KUKA KRL program: MyProgram_049().src

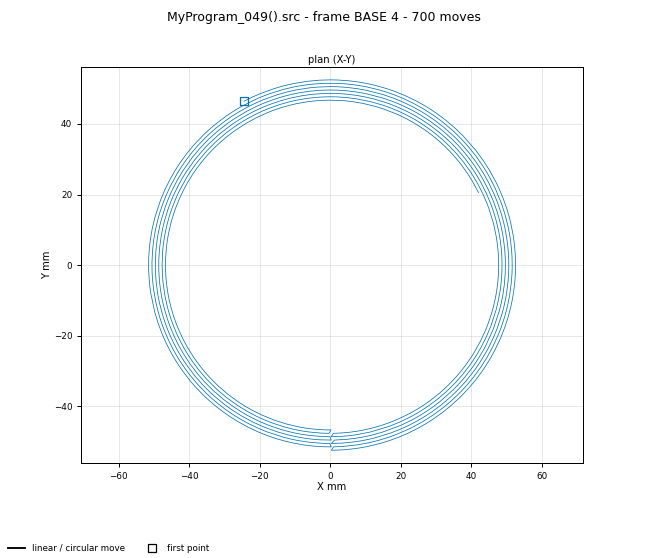
[picture p0: tool path of MyProgram_049().src in frame BASE 4, 700 of 700 moves have a stored position in this frame; points joined in program order, loops and branches not executed]
&ACCESS RVP
&REL 1
&PARAM TEMPLATE = C:\KRC\Roboter\Template\vorgabe
&PARAM EDITMASK = *
DEF MyProgram_049()
; ---- Setting reference (Base) ----
$BASE = BASE_DATA[4]

; --------------------------
; ---- Setting tool (TCP) ----
$TOOL = TOOL_DATA[3]
; --------------------------

$VEL.CP = VEL_APROX_PRINT
Startdeposition()
$VEL.CP = VEL_PRINT
LIN {X -24.4251,Y 46.489,Z 66,A 110.3298,B 24.8528,C -2.799,E1 24.9276,E2 -26.6779} C_DIS
LIN {X -22.2975,Y 47.5462,Z 66,A 107.8402,B 24.8522,C -2.8046,E1 24.9338,E2 -24.1953} C_DIS
LIN {X -20.0444,Y 48.539,Z 66,A 104.5324,B 24.8529,C -2.7984,E1 24.9424,E2 -20.8649} C_DIS
LIN {X -15.8817,Y 50.0558,Z 66,A 100.3319,B 24.8512,C -2.8146,E1 24.9534,E2 -16.695} C_DIS
LIN {X -13.4432,Y 50.7654,Z 66,A 97.3988,B 24.8512,C -2.8147,E1 24.9613,E2 -13.7577} C_DIS
LIN {X -10.7407,Y 51.4051,Z 66,A 93.9354,B 24.8517,C -2.8101,E1 24.9708,E2 -10.279} C_DIS
LIN {X -6.5682,Y 52.1029,Z 66,A 89.9124,B 24.8503,C -2.8232,E1 24.9818,E2 -6.2837} C_DIS
LIN {X -3.1559,Y 52.4207,Z 66,A 85.9853,B 24.8504,C -2.8216,E1 24.9927,E2 -2.3511} C_DIS
LIN {X 0.019,Y 52.5158,Z 66,A 82.4303,B 24.8505,C -2.8209,E1 25.0027,E2 1.2058} C_DIS
LIN {X 2.2082,Y 52.4685,Z 66,A 79.9006,B 24.8507,C -2.8187,E1 25.0097,E2 3.7403} C_DIS
LIN {X 5.4247,Y 52.234,Z 66,A 76.6583,B 24.8503,C -2.8233,E1 25.0187,E2 6.9698} C_DIS
LIN {X 8.0055,Y 51.9012,Z 66,A 73.774,B 24.8504,C -2.8218,E1 25.0267,E2 9.8551} C_DIS
LIN {X 10.5647,Y 51.4413,Z 66,A 71.0397,B 24.8504,C -2.8225,E1 25.0342,E2 12.5846} C_DIS
LIN {X 12.7838,Y 50.935,Z 66,A 68.4031,B 24.8508,C -2.8183,E1 25.0414,E2 15.2272} C_DIS
LIN {X 15.987,Y 50.0225,Z 66,A 65.1391,B 24.8503,C -2.8226,E1 25.0501,E2 18.4755} C_DIS
LIN {X 18.0888,Y 49.3014,Z 66,A 62.3939,B 24.8512,C -2.8145,E1 25.0573,E2 21.2343} C_DIS
LIN {X 21.2443,Y 48.026,Z 66,A 58.6048,B 24.8518,C -2.8092,E1 25.0671,E2 25.0269} C_DIS
LIN {X 24.339,Y 46.5341,Z 66,A 55.5963,B 24.8507,C -2.8188,E1 25.0745,E2 28.0049} C_DIS
LIN {X 26.498,Y 45.3396,Z 66,A 52.1536,B 24.8527,C -2.8006,E1 25.083,E2 31.4803} C_DIS
LIN {X 28.6427,Y 44.0153,Z 66,A 49.6719,B 24.8526,C -2.8016,E1 25.0888,E2 33.9516} C_DIS
LIN {X 30.216,Y 42.9521,Z 66,A 47.4699,B 24.8532,C -2.7957,E1 25.0939,E2 36.1601} C_DIS
LIN {X 32.4632,Y 41.2792,Z 66,A 44.4209,B 24.8537,C -2.7905,E1 25.1006,E2 39.2102} C_DIS
LIN {X 35.455,Y 38.7397,Z 66,A 40.2431,B 24.8544,C -2.7844,E1 25.1094,E2 43.3862} C_DIS
LIN {X 37.586,Y 36.6762,Z 66,A 36.7099,B 24.8557,C -2.7718,E1 25.1164,E2 46.9343} C_DIS
LIN {X 41.2065,Y 32.5552,Z 66,A 31.7321,B 24.855,C -2.7786,E1 25.1255,E2 51.8734} C_DIS
LIN {X 43.4466,Y 29.4994,Z 66,A 26.8425,B 24.8576,C -2.7532,E1 25.1335,E2 56.7995} C_DIS
LIN {X 45.1779,Y 26.7727,Z 66,A 23.6494,B 24.8579,C -2.7509,E1 25.1382,E2 59.9819} C_DIS
LIN {X 47.1008,Y 23.2237,Z 66,A 19.3403,B 24.8589,C -2.741,E1 25.1439,E2 64.2916} C_DIS
LIN {X 47.7499,Y 21.8578,Z 66,A 16.8923,B 24.8611,C -2.72,E1 25.1467,E2 66.7761} C_DIS
LIN {X 48.9324,Y 19.0647,Z 66,A 14.0783,B 24.861,C -2.7208,E1 25.1497,E2 69.5726} C_DIS
LIN {X 50.0654,Y 15.8514,Z 66,A 10.5617,B 24.8616,C -2.7142,E1 25.1528,E2 73.0851} C_DIS
LIN {X 50.6849,Y 13.7421,Z 66,A 8.1164,B 24.8625,C -2.7061,E1 25.1547,E2 75.5356} C_DIS
LIN {X 51.1251,Y 12.0025,Z 66,A 5.8316,B 24.8638,C -2.6933,E1 25.1562,E2 77.8373} C_DIS
LIN {X 51.8393,Y 8.4,Z 66,A 2.4748,B 24.8636,C -2.6947,E1 25.1579,E2 81.1712} C_DIS
LIN {X 52.1505,Y 6.1764,Z 66,A -0.4769,B 24.8655,C -2.6766,E1 25.1589,E2 84.1483} C_DIS
LIN {X 52.4193,Y 3.1759,Z 66,A -3.9297,B 24.8669,C -2.6628,E1 25.1596,E2 87.6132} C_DIS
LIN {X 52.5126,Y -0.462,Z 66,A -7.4944,B 24.8672,C -2.6589,E1 25.1597,E2 91.1659} C_DIS
LIN {X 52.4191,Y -3.1656,Z 66,A -10.1321,B 24.8675,C -2.6562,E1 25.1594,E2 93.7943} C_DIS
LIN {X 52.2992,Y -4.7558,Z 66,A -12.1864,B 24.8687,C -2.6441,E1 25.1589,E2 95.8651} C_DIS
LIN {X 51.9991,Y -7.3421,Z 66,A -14.8639,B 24.8693,C -2.6386,E1 25.158,E2 98.5398} C_DIS
LIN {X 51.6388,Y -9.5543,Z 66,A -17.2732,B 24.87,C -2.6316,E1 25.1568,E2 100.9514} C_DIS
LIN {X 51.2544,Y -11.4372,Z 66,A -19.8065,B 24.8715,C -2.6159,E1 25.1553,E2 103.5072} C_DIS
LIN {X 50.3186,Y -15.0287,Z 66,A -23.5172,B 24.8721,C -2.6105,E1 25.1526,E2 107.2093} C_DIS
LIN {X 49.5084,Y -17.5135,Z 66,A -26.3955,B 24.873,C -2.6012,E1 25.15,E2 110.0933} C_DIS
LIN {X 48.4841,Y -20.1769,Z 66,A -29.1133,B 24.873,C -2.6002,E1 25.1472,E2 112.7985} C_DIS
LIN {X 47.9293,Y -21.4606,Z 66,A -31.0442,B 24.8743,C -2.5872,E1 25.145,E2 114.7498} C_DIS
LIN {X 46.529,Y -24.3487,Z 66,A -34.3749,B 24.875,C -2.5805,E1 25.1408,E2 118.0783} C_DIS
LIN {X 45.286,Y -26.5899,Z 66,A -37.4931,B 24.8764,C -2.5659,E1 25.1365,E2 121.2151} C_DIS
LIN {X 43.7354,Y -29.0701,Z 66,A -40.2741,B 24.8764,C -2.5655,E1 25.1323,E2 123.9829} C_DIS
LIN {X 42.5013,Y -30.8459,Z 66,A -42.7432,B 24.8773,C -2.5569,E1 25.1283,E2 126.4603} C_DIS
LIN {X 41.2562,Y -32.4924,Z 66,A -45.0593,B 24.878,C -2.5497,E1 25.1243,E2 128.7827} C_DIS
LIN {X 39.4232,Y -34.6939,Z 66,A -48.1201,B 24.8786,C -2.5431,E1 25.1188,E2 131.8452} C_DIS
LIN {X 36.7356,Y -37.5281,Z 66,A -52.9038,B 24.8806,C -2.5222,E1 25.1093,E2 136.6578} C_DIS
LIN {X 33.9294,Y -40.083,Z 66,A -56.4666,B 24.8804,C -2.5246,E1 25.1019,E2 140.2009} C_DIS
LIN {X 31.7525,Y -41.829,Z 66,A -59.5227,B 24.881,C -2.5179,E1 25.0952,E2 143.2616} C_DIS
LIN {X 29.2965,Y -43.5834,Z 66,A -62.5914,B 24.8812,C -2.5158,E1 25.0882,E2 146.3246} C_DIS
LIN {X 27.1565,Y -44.9481,Z 66,A -65.8284,B 24.8825,C -2.5014,E1 25.0804,E2 149.5854} C_DIS
LIN {X 24.6543,Y -46.3684,Z 66,A -68.7154,B 24.8825,C -2.501,E1 25.0734,E2 152.4651} C_DIS
LIN {X 22.1208,Y -47.6287,Z 66,A -71.7781,B 24.883,C -2.4967,E1 25.0657,E2 155.5301} C_DIS
LIN {X 19.4367,Y -48.7857,Z 66,A -74.9858,B 24.8835,C -2.4918,E1 25.0574,E2 158.7419} C_DIS
LIN {X 16.7705,Y -49.7651,Z 66,A -78.018,B 24.8837,C -2.4891,E1 25.0494,E2 161.7742} C_DIS
LIN {X 14.1882,Y -50.5619,Z 66,A -81.1897,B 24.8844,C -2.4816,E1 25.0409,E2 164.9583} C_DIS
LIN {X 10.6217,Y -51.4296,Z 66,A -84.7511,B 24.884,C -2.4863,E1 25.0312,E2 168.5038} C_DIS
LIN {X 8.5887,Y -51.8079,Z 66,A -87.0096,B 24.8841,C -2.4845,E1 25.025,E2 170.764} C_DIS
LIN {X 6.6367,Y -52.0936,Z 66,A -89.3786,B 24.8846,C -2.4791,E1 25.0184,E2 173.144} C_DIS
LIN {X 3.7845,Y -52.379,Z 66,A -92.2753,B 24.8844,C -2.4818,E1 25.0104,E2 176.0327} C_DIS
LIN {X 1.9687,Y -52.4779,Z 66,A -94.4349,B 24.8848,C -2.4778,E1 25.0043,E2 178.201} C_DIS
LIN {X 0.2751,Y -52.5115,Z 66,A -95.8459,B 24.8841,C -2.4854,E1 25.0004,E2 179.5939} C_DIS
Enddeposition()
LIN {X 0.2751,Y -52.5115,Z 66,A -95.8459,B 24.8841,C -2.4854,E1 25.0004,E2 179.5939} C_DIS
Startdeposition()
$VEL.CP = VEL_PRINT
LIN {X 0.9003,Y -51.5477,Z 66,A -94.1918,B 24.8808,C -2.5197,E1 25.0053,E2 177.8585} C_DIS
LIN {X 3.5763,Y -51.4318,Z 66,A -90.9185,B 24.8802,C -2.5264,E1 25.0144,E2 174.5705} C_DIS
LIN {X 7.7801,Y -50.9656,Z 66,A -86.3222,B 24.8801,C -2.5274,E1 25.0272,E2 169.9756} C_DIS
LIN {X 10.8144,Y -50.4088,Z 66,A -83.1139,B 24.8802,C -2.5261,E1 25.0359,E2 166.7742} C_DIS
LIN {X 13.4755,Y -49.7634,Z 66,A -79.8609,B 24.8795,C -2.5332,E1 25.0448,E2 163.5094} C_DIS
LIN {X 16.9849,Y -48.6775,Z 66,A -76.2382,B 24.8799,C -2.5292,E1 25.0543,E2 159.903} C_DIS
LIN {X 18.7561,Y -48.0231,Z 66,A -73.5337,B 24.8785,C -2.5438,E1 25.0615,E2 157.1698} C_DIS
LIN {X 22.8223,Y -46.2294,Z 66,A -69.2117,B 24.879,C -2.5391,E1 25.0724,E2 152.8697} C_DIS
LIN {X 26.1375,Y -44.4389,Z 66,A -64.44,B 24.8772,C -2.558,E1 25.0841,E2 148.0673} C_DIS
LIN {X 29.0142,Y -42.6165,Z 66,A -60.8596,B 24.8769,C -2.5612,E1 25.0924,E2 144.4913} C_DIS
LIN {X 31.4014,Y -40.8897,Z 66,A -57.7626,B 24.8765,C -2.5644,E1 25.0993,E2 141.3978} C_DIS
LIN {X 33.5879,Y -39.114,Z 66,A -54.305,B 24.8752,C -2.5779,E1 25.1067,E2 137.9216} C_DIS
LIN {X 36.0946,Y -36.8134,Z 66,A -51.1243,B 24.8756,C -2.5744,E1 25.1131,E2 134.7622} C_DIS
LIN {X 37.5261,Y -35.3525,Z 66,A -48.8389,B 24.875,C -2.5802,E1 25.1176,E2 132.473} C_DIS
LIN {X 38.6864,Y -34.0796,Z 66,A -46.7252,B 24.8741,C -2.5891,E1 25.1215,E2 130.3477} C_DIS
LIN {X 40.4912,Y -31.9136,Z 66,A -43.3418,B 24.8728,C -2.6024,E1 25.1275,E2 126.9485} C_DIS
LIN {X 42.5712,Y -29.0816,Z 66,A -39.7719,B 24.8725,C -2.6059,E1 25.1332,E2 123.3876} C_DIS
LIN {X 44.2529,Y -26.4525,Z 66,A -35.946,B 24.8708,C -2.6231,E1 25.1389,E2 119.5405} C_DIS
LIN {X 45.9151,Y -23.4477,Z 66,A -32.0497,B 24.8695,C -2.6358,E1 25.1439,E2 115.6348} C_DIS
LIN {X 47.7204,Y -19.5136,Z 66,A -27.9551,B 24.8696,C -2.635,E1 25.1485,E2 111.5644} C_DIS
LIN {X 48.4134,Y -17.7236,Z 66,A -25.385,B 24.8681,C -2.6507,E1 25.151,E2 108.9716} C_DIS
LIN {X 49.5223,Y -14.3369,Z 66,A -21.6876,B 24.8674,C -2.6573,E1 25.1541,E2 105.2797} C_DIS
LIN {X 50.228,Y -11.6257,Z 66,A -18.6184,B 24.8665,C -2.666,E1 25.1561,E2 102.2076} C_DIS
LIN {X 50.826,Y -8.6459,Z 66,A -14.7246,B 24.8644,C -2.6876,E1 25.1581,E2 98.2856} C_DIS
LIN {X 51.3544,Y -4.5536,Z 66,A -10.799,B 24.8644,C -2.688,E1 25.1593,E2 94.3822} C_DIS
LIN {X 51.5107,Y -2.1502,Z 66,A -8.2787,B 24.8638,C -2.6931,E1 25.1597,E2 91.8647} C_DIS
LIN {X 51.5542,Y -0.2569,Z 66,A -6.0511,B 24.8629,C -2.7024,E1 25.1597,E2 89.6285} C_DIS
LIN {X 51.5056,Y 2.2745,Z 66,A -3.2025,B 24.8619,C -2.7119,E1 25.1595,E2 86.7742} C_DIS
LIN {X 51.3916,Y 4.1131,Z 66,A -0.9354,B 24.8608,C -2.7229,E1 25.159,E2 84.4945} C_DIS
LIN {X 51.0902,Y 6.9164,Z 66,A 1.7719,B 24.8607,C -2.7237,E1 25.1581,E2 81.8015} C_DIS
LIN {X 50.8314,Y 8.6131,Z 66,A 3.8539,B 24.8597,C -2.7332,E1 25.1572,E2 79.7091} C_DIS
LIN {X 50.3222,Y 11.2104,Z 66,A 6.7142,B 24.859,C -2.7404,E1 25.1556,E2 76.8485} C_DIS
LIN {X 49.3934,Y 14.7756,Z 66,A 10.4,B 24.8586,C -2.7441,E1 25.1529,E2 73.1752} C_DIS
LIN {X 48.4755,Y 17.5543,Z 66,A 14.1514,B 24.8565,C -2.7639,E1 25.1495,E2 69.398} C_DIS
LIN {X 46.7087,Y 21.8246,Z 66,A 18.872,B 24.8559,C -2.7697,E1 25.1443,E2 64.6895} C_DIS
LIN {X 45.3442,Y 24.5338,Z 66,A 22.6057,B 24.8542,C -2.7863,E1 25.1395,E2 60.9363} C_DIS
LIN {X 44.433,Y 26.1481,Z 66,A 24.7421,B 24.8534,C -2.7932,E1 25.1365,E2 58.7945} C_DIS
LIN {X 43.147,Y 28.2202,Z 66,A 27.0364,B 24.8536,C -2.7916,E1 25.1331,E2 56.5156} C_DIS
LIN {X 41.2251,Y 30.9597,Z 66,A 30.7286,B 24.8527,C -2.8002,E1 25.1271,E2 52.8212} C_DIS
LIN {X 39.1193,Y 33.5811,Z 66,A 34.717,B 24.8513,C -2.8138,E1 25.12,E2 48.8189} C_DIS
LIN {X 37.8892,Y 34.9634,Z 66,A 36.9383,B 24.8504,C -2.8216,E1 25.1158,E2 46.5889} C_DIS
LIN {X 35.6984,Y 37.1974,Z 66,A 39.9299,B 24.8507,C -2.8191,E1 25.1099,E2 43.6157} C_DIS
LIN {X 34.4399,Y 38.3652,Z 66,A 42.4096,B 24.8491,C -2.8342,E1 25.1047,E2 41.1102} C_DIS
LIN {X 31.7707,Y 40.6041,Z 66,A 45.9402,B 24.8491,C -2.8346,E1 25.0971,E2 37.5922} C_DIS
LIN {X 29.6449,Y 42.1811,Z 66,A 49.8098,B 24.8466,C -2.8576,E1 25.0882,E2 33.6813} C_DIS
LIN {X 26.515,Y 44.2153,Z 66,A 53.6181,B 24.8466,C -2.8571,E1 25.0792,E2 29.8863} C_DIS
LIN {X 23.289,Y 45.996,Z 66,A 57.5115,B 24.8465,C -2.8585,E1 25.0695,E2 26.0006} C_DIS
LIN {X 20.4247,Y 47.3378,Z 66,A 60.2231,B 24.8477,C -2.8472,E1 25.0627,E2 23.3225} C_DIS
LIN {X 17.9374,Y 48.3348,Z 66,A 63.0896,B 24.8477,C -2.848,E1 25.0553,E2 20.4604} C_DIS
LIN {X 16.2204,Y 48.9381,Z 66,A 65.7948,B 24.8461,C -2.8623,E1 25.0481,E2 17.7265} C_DIS
LIN {X 13.8269,Y 49.6664,Z 66,A 68.6101,B 24.8458,C -2.8649,E1 25.0405,E2 14.9099} C_DIS
LIN {X 10.3647,Y 50.5033,Z 66,A 72.1007,B 24.8465,C -2.8583,E1 25.0311,E2 11.4396} C_DIS
LIN {X 8.5617,Y 50.84,Z 66,A 74.5418,B 24.8456,C -2.8663,E1 25.0243,E2 8.9822} C_DIS
LIN {X 6.0982,Y 51.1941,Z 66,A 76.9306,B 24.8463,C -2.8601,E1 25.0177,E2 6.61} C_DIS
LIN {X 3.8919,Y 51.4091,Z 66,A 79.7094,B 24.8457,C -2.8659,E1 25.01,E2 3.819} C_DIS
LIN {X 1.3954,Y 51.537,Z 66,A 82.9501,B 24.8448,C -2.8739,E1 25.0009,E2 0.56} C_DIS
LIN {X -1.7915,Y 51.5249,Z 66,A 85.5886,B 24.8466,C -2.8571,E1 24.9936,E2 -2.0388} C_DIS
LIN {X -5.366,Y 51.2759,Z 66,A 89.6135,B 24.8467,C -2.8561,E1 24.9824,E2 -6.063} C_DIS
LIN {X -8.0268,Y 50.9274,Z 66,A 93.0737,B 24.8461,C -2.8624,E1 24.9728,E2 -9.5409} C_DIS
LIN {X -10.5231,Y 50.4708,Z 66,A 96.2084,B 24.8457,C -2.8654,E1 24.9642,E2 -12.6865} C_DIS
LIN {X -13.6315,Y 49.7212,Z 66,A 99.3494,B 24.8469,C -2.855,E1 24.9558,E2 -15.8073} C_DIS
LIN {X -17.5748,Y 48.468,Z 66,A 104.4749,B 24.8465,C -2.8583,E1 24.9422,E2 -20.9502} C_DIS
LIN {X -20.2955,Y 47.3931,Z 66,A 108.0024,B 24.8465,C -2.8583,E1 24.9331,E2 -24.4858} C_DIS
LIN {X -25.0049,Y 45.0864,Z 66,A 112.8761,B 24.8492,C -2.8334,E1 24.9211,E2 -29.3134} C_DIS
LIN {X -26.9453,Y 43.9537,Z 66,A 115.6363,B 24.8492,C -2.8331,E1 24.9145,E2 -32.0815} C_DIS
LIN {X -29.4226,Y 42.3358,Z 66,A 119.2758,B 24.8492,C -2.8324,E1 24.906,E2 -35.7313} C_DIS
LIN {X -33.0763,Y 39.5474,Z 66,A 123.7719,B 24.8515,C -2.8121,E1 24.8962,E2 -40.1955} C_DIS
LIN {X -35.6913,Y 37.2036,Z 66,A 128.3068,B 24.8514,C -2.813,E1 24.8869,E2 -44.751} C_DIS
LIN {X -38.5307,Y 34.2544,Z 66,A 133.0331,B 24.8522,C -2.8045,E1 24.878,E2 -49.478} C_DIS
LIN {X -40.5386,Y 31.8536,Z 66,A 135.842,B 24.8543,C -2.7854,E1 24.8731,E2 -52.2543} C_DIS
LIN {X -42.42,Y 29.3015,Z 66,A 139.848,B 24.8545,C -2.7833,E1 24.8666,E2 -56.2747} C_DIS
LIN {X -44.0768,Y 26.7441,Z 66,A 142.8215,B 24.8561,C -2.7677,E1 24.8622,E2 -59.2262} C_DIS
LIN {X -45.4139,Y 24.4051,Z 66,A 145.9986,B 24.8567,C -2.7619,E1 24.8579,E2 -62.406} C_DIS
LIN {X -46.9173,Y 21.372,Z 66,A 150.1658,B 24.8572,C -2.7569,E1 24.8529,E2 -66.584} C_DIS
LIN {X -48.2045,Y 18.2848,Z 66,A 154.0614,B 24.8581,C -2.7484,E1 24.8489,E2 -70.4811} C_DIS
LIN {X -49.752,Y 13.5185,Z 66,A 158.8731,B 24.861,C -2.7202,E1 24.845,E2 -75.2529} C_DIS
LIN {X -50.4731,Y 10.5091,Z 66,A 162.8027,B 24.8614,C -2.7167,E1 24.8426,E2 -79.1972} C_DIS
LIN {X -51.0003,Y 7.5441,Z 66,A 166.0072,B 24.8627,C -2.7041,E1 24.8412,E2 -82.3907} C_DIS
LIN {X -51.3369,Y 4.7467,Z 66,A 169.109,B 24.8637,C -2.6938,E1 24.8403,E2 -85.4864} C_DIS
LIN {X -51.5176,Y 1.9972,Z 66,A 172.2934,B 24.8645,C -2.6859,E1 24.8398,E2 -88.6712} C_DIS
LIN {X -51.5363,Y -1.423,Z 66,A 176.3078,B 24.8654,C -2.6772,E1 24.84,E2 -92.6888} C_DIS
LIN {X -51.3057,Y -5.0748,Z 66,A -179.8668,B 24.867,C -2.6609,E1 24.8408,E2 -96.4984} C_DIS
LIN {X -50.9516,Y -7.8706,Z 66,A -175.9049,B 24.8668,C -2.6636,E1 24.8424,E2 -100.4903} C_DIS
LIN {X -49.8182,Y -13.2732,Z 66,A -170.0005,B 24.869,C -2.6417,E1 24.8462,E2 -106.3767} C_DIS
LIN {X -48.8876,Y -16.3714,Z 66,A -166.6975,B 24.8704,C -2.6267,E1 24.8491,E2 -109.6631} C_DIS
LIN {X -47.6249,Y -19.7451,Z 66,A -163.316,B 24.8725,C -2.606,E1 24.8524,E2 -113.014} C_DIS
LIN {X -46.6955,Y -21.8527,Z 66,A -160.2524,B 24.8725,C -2.6065,E1 24.856,E2 -116.0955} C_DIS
LIN {X -45.6573,Y -23.9461,Z 66,A -158.0125,B 24.8737,C -2.5941,E1 24.8588,E2 -118.3177} C_DIS
LIN {X -44.7271,Y -25.6417,Z 66,A -155.7934,B 24.8741,C -2.5895,E1 24.8618,E2 -120.5374} C_DIS
LIN {X -43.408,Y -27.8164,Z 66,A -152.4793,B 24.8741,C -2.5897,E1 24.8668,E2 -123.8691} C_DIS
LIN {X -41.9889,Y -29.9156,Z 66,A -149.4961,B 24.8745,C -2.5854,E1 24.8716,E2 -126.8567} C_DIS
LIN {X -39.593,Y -33.0214,Z 66,A -145.8008,B 24.8765,C -2.5649,E1 24.878,E2 -130.5204} C_DIS
LIN {X -38.3674,Y -34.4377,Z 66,A -143.7078,B 24.8769,C -2.5605,E1 24.8818,E2 -132.6122} C_DIS
LIN {X -36.1762,Y -36.7328,Z 66,A -140.2072,B 24.8777,C -2.5527,E1 24.8886,E2 -136.1092} C_DIS
LIN {X -35.0907,Y -37.7718,Z 66,A -138.1632,B 24.8774,C -2.5553,E1 24.8928,E2 -138.1678} C_DIS
LIN {X -32.6423,Y -39.9067,Z 66,A -134.4662,B 24.8779,C -2.55,E1 24.9007,E2 -141.8664} C_DIS
LIN {X -30.4324,Y -41.6158,Z 66,A -131.5674,B 24.8788,C -2.5413,E1 24.9071,E2 -144.7549} C_DIS
LIN {X -28.4555,Y -42.9919,Z 66,A -128.7353,B 24.8789,C -2.5396,E1 24.9137,E2 -147.5924} C_DIS
LIN {X -26.4079,Y -44.2794,Z 66,A -126.2831,B 24.8797,C -2.5319,E1 24.9195,E2 -150.0337} C_DIS
LIN {X -23.2124,Y -46.0349,Z 66,A -121.3528,B 24.8788,C -2.5414,E1 24.9318,E2 -155.0005} C_DIS
LIN {X -20.4483,Y -47.3276,Z 66,A -118.54,B 24.88,C -2.528,E1 24.9389,E2 -157.7879} C_DIS
LIN {X -17.6341,Y -48.446,Z 66,A -115.4427,B 24.8808,C -2.5203,E1 24.9469,E2 -160.8736} C_DIS
LIN {X -15.1235,Y -49.288,Z 66,A -112.0558,B 24.8802,C -2.5258,E1 24.956,E2 -164.2795} C_DIS
LIN {X -12.6811,Y -49.972,Z 66,A -109.7551,B 24.8813,C -2.5151,E1 24.9621,E2 -166.5583} C_DIS
LIN {X -10.845,Y -50.4023,Z 66,A -107.5392,B 24.8812,C -2.5162,E1 24.9682,E2 -168.7797} C_DIS
LIN {X -7.6088,Y -50.992,Z 66,A -103.1403,B 24.88,C -2.5284,E1 24.9804,E2 -173.2116} C_DIS
LIN {X -4.5201,Y -51.3573,Z 66,A -100.1449,B 24.8808,C -2.5198,E1 24.9887,E2 -176.1882} C_DIS
LIN {X -1.8786,Y -51.5219,Z 66,A -97.4426,B 24.8812,C -2.5157,E1 24.9962,E2 -178.8814} C_DIS
LIN {X 0.2651,Y -51.5544,Z 66,A -95.3508,B 24.8817,C -2.5109,E1 25.002,E2 -180.9619} C_DIS
Enddeposition()
LIN {X 0.2651,Y -51.5544,Z 66,A -95.3508,B 24.8817,C -2.5109,E1 25.002,E2 -180.9619} C_DIS
Startdeposition()
$VEL.CP = VEL_PRINT
LIN {X -0.1922,Y -50.5965,Z 66,A -96.6326,B 24.8814,C -2.5138,E1 24.9984,E2 -179.6869} C_DIS
LIN {X -2.0456,Y -50.5555,Z 66,A -99.5612,B 24.8828,C -2.4992,E1 24.9902,E2 -176.7231} C_DIS
LIN {X -5.4618,Y -50.301,Z 66,A -103.2186,B 24.8824,C -2.5032,E1 24.98,E2 -173.0734} C_DIS
LIN {X -8.8334,Y -49.8198,Z 66,A -106.7107,B 24.8817,C -2.5104,E1 24.9704,E2 -169.5953} C_DIS
LIN {X -11.0833,Y -49.368,Z 66,A -109.2933,B 24.8816,C -2.5118,E1 24.9634,E2 -167.013} C_DIS
LIN {X -13.2229,Y -48.8384,Z 66,A -112.4248,B 24.8824,C -2.5028,E1 24.9548,E2 -163.8552} C_DIS
LIN {X -17.944,Y -47.3079,Z 66,A -117.5123,B 24.8812,C -2.516,E1 24.9415,E2 -158.7895} C_DIS
LIN {X -20.1645,Y -46.4047,Z 66,A -120.8148,B 24.8818,C -2.5094,E1 24.9329,E2 -155.4635} C_DIS
LIN {X -23.3404,Y -44.8918,Z 66,A -124.138,B 24.8804,C -2.5247,E1 24.9247,E2 -152.1679} C_DIS
LIN {X -25.7018,Y -43.5828,Z 66,A -127.406,B 24.8803,C -2.5255,E1 24.9168,E2 -148.8923} C_DIS
LIN {X -27.975,Y -42.16,Z 66,A -130.1506,B 24.8794,C -2.5347,E1 24.9103,E2 -146.1607} C_DIS
LIN {X -29.9616,Y -40.7719,Z 66,A -133.2367,B 24.8794,C -2.5339,E1 24.9033,E2 -143.062} C_DIS
LIN {X -31.7244,Y -39.4161,Z 66,A -135.4138,B 24.8785,C -2.5436,E1 24.8986,E2 -140.9} C_DIS
LIN {X -33.4661,Y -37.9489,Z 66,A -138.1725,B 24.8783,C -2.5457,E1 24.8927,E2 -138.1355} C_DIS
LIN {X -35.1369,Y -36.4065,Z 66,A -141.5564,B 24.879,C -2.5388,E1 24.8859,E2 -134.7211} C_DIS
LIN {X -37.554,Y -33.9083,Z 66,A -145.2942,B 24.8779,C -2.5502,E1 24.8788,E2 -130.9942} C_DIS
LIN {X -39.8163,Y -31.2208,Z 66,A -148.7061,B 24.8762,C -2.5677,E1 24.8728,E2 -127.6081} C_DIS
LIN {X -41.5359,Y -28.893,Z 66,A -151.9555,B 24.8754,C -2.5761,E1 24.8675,E2 -124.3629} C_DIS
LIN {X -42.8846,Y -26.8506,Z 66,A -154.7636,B 24.8748,C -2.5825,E1 24.8633,E2 -121.556} C_DIS
LIN {X -43.9001,Y -25.156,Z 66,A -156.7354,B 24.8738,C -2.5922,E1 24.8605,E2 -119.5971} C_DIS
LIN {X -44.8198,Y -23.4779,Z 66,A -159.1161,B 24.8736,C -2.5949,E1 24.8574,E2 -117.2102} C_DIS
LIN {X -45.8817,Y -21.3285,Z 66,A -162.0242,B 24.8731,C -2.5996,E1 24.8539,E2 -114.2975} C_DIS
LIN {X -46.887,Y -19.0171,Z 66,A -164.8375,B 24.8723,C -2.6082,E1 24.8508,E2 -111.4892} C_DIS
LIN {X -47.7932,Y -16.6083,Z 66,A -167.3954,B 24.871,C -2.6216,E1 24.8484,E2 -108.9489} C_DIS
LIN {X -48.2308,Y -15.2911,Z 66,A -169.2342,B 24.8709,C -2.6224,E1 24.8468,E2 -107.1016} C_DIS
LIN {X -48.8214,Y -13.2849,Z 66,A -171.7035,B 24.8703,C -2.628,E1 24.8449,E2 -104.6313} C_DIS
LIN {X -49.475,Y -10.5951,Z 66,A -175.0294,B 24.8696,C -2.6348,E1 24.8429,E2 -101.3021} C_DIS
LIN {X -50.1285,Y -6.873,Z 66,A -179.2581,B 24.8683,C -2.6486,E1 24.841,E2 -97.0813} C_DIS
LIN {X -50.4189,Y -4.2446,Z 66,A 178.1838,B 24.8667,C -2.664,E1 24.8403,E2 -94.5447} C_DIS
LIN {X -50.5525,Y -2.1183,Z 66,A 175.2997,B 24.8667,C -2.665,E1 24.8398,E2 -91.6455} C_DIS
LIN {X -50.5929,Y 0.6544,Z 66,A 171.6752,B 24.8663,C -2.6682,E1 24.8398,E2 -88.0069} C_DIS
LIN {X -50.4224,Y 4.2008,Z 66,A 168.1736,B 24.8643,C -2.688,E1 24.8405,E2 -84.5316} C_DIS
LIN {X -50.0849,Y 7.1793,Z 66,A 164.555,B 24.8635,C -2.6956,E1 24.8418,E2 -80.9095} C_DIS
LIN {X -49.6027,Y 9.9792,Z 66,A 160.9628,B 24.863,C -2.7005,E1 24.8437,E2 -77.3078} C_DIS
LIN {X -48.906,Y 12.972,Z 66,A 158.0771,B 24.8611,C -2.7194,E1 24.8456,E2 -74.4505} C_DIS
LIN {X -48.3534,Y 14.8983,Z 66,A 155.6256,B 24.8607,C -2.7239,E1 24.8476,E2 -71.9955} C_DIS
LIN {X -47.4417,Y 17.5875,Z 66,A 152.5704,B 24.8594,C -2.7359,E1 24.8504,E2 -68.9516} C_DIS
LIN {X -46.6479,Y 19.5962,Z 66,A 149.7953,B 24.8591,C -2.7386,E1 24.8533,E2 -66.1675} C_DIS
LIN {X -45.3426,Y 22.452,Z 66,A 146.0658,B 24.8583,C -2.7465,E1 24.8578,E2 -62.4368} C_DIS
LIN {X -43.4081,Y 25.9954,Z 66,A 141.8799,B 24.8564,C -2.7649,E1 24.8636,E2 -58.273} C_DIS
LIN {X -42.134,Y 28.0141,Z 66,A 139.1728,B 24.8556,C -2.7723,E1 24.8677,E2 -55.5698} C_DIS
LIN {X -40.7058,Y 30.0518,Z 66,A 136.1782,B 24.8551,C -2.7772,E1 24.8725,E2 -52.5726} C_DIS
LIN {X -39.2355,Y 31.9472,Z 66,A 133.6637,B 24.8541,C -2.7872,E1 24.8769,E2 -50.0699} C_DIS
LIN {X -37.5356,Y 33.9286,Z 66,A 130.4034,B 24.8538,C -2.7901,E1 24.8829,E2 -46.8021} C_DIS
LIN {X -35.3455,Y 36.2047,Z 66,A 126.6629,B 24.8531,C -2.7962,E1 24.8903,E2 -43.0603} C_DIS
LIN {X -33.453,Y 37.9602,Z 66,A 124.2101,B 24.8517,C -2.8097,E1 24.8953,E2 -40.6297} C_DIS
LIN {X -31.9684,Y 39.2184,Z 66,A 121.9246,B 24.8513,C -2.8132,E1 24.9002,E2 -38.3439} C_DIS
LIN {X -29.989,Y 40.7519,Z 66,A 118.8227,B 24.8511,C -2.8151,E1 24.9071,E2 -35.2353} C_DIS
LIN {X -27.9743,Y 42.1604,Z 66,A 116.3188,B 24.8501,C -2.8246,E1 24.9129,E2 -32.7459} C_DIS
LIN {X -25.7013,Y 43.5831,Z 66,A 112.9533,B 24.8501,C -2.8251,E1 24.9209,E2 -29.3711} C_DIS
LIN {X -22.6142,Y 45.2616,Z 66,A 108.6196,B 24.8499,C -2.8262,E1 24.9317,E2 -25.0281} C_DIS
LIN {X -19.5958,Y 46.6481,Z 66,A 104.724,B 24.8496,C -2.8295,E1 24.9417,E2 -21.1312} C_DIS
LIN {X -14.999,Y 48.3225,Z 66,A 100.0446,B 24.8474,C -2.8497,E1 24.9539,E2 -16.491} C_DIS
LIN {X -12.0934,Y 49.1299,Z 66,A 96.0651,B 24.848,C -2.8441,E1 24.9647,E2 -12.4921} C_DIS
LIN {X -9.4929,Y 49.6983,Z 66,A 93.5946,B 24.8468,C -2.8554,E1 24.9714,E2 -10.0455} C_DIS
LIN {X -5.9552,Y 50.2452,Z 66,A 89.6571,B 24.8463,C -2.8599,E1 24.9823,E2 -6.1156} C_DIS
LIN {X -3.6552,Y 50.4652,Z 66,A 86.3052,B 24.8475,C -2.8489,E1 24.9917,E2 -2.736} C_DIS
LIN {X -0.0826,Y 50.5969,Z 66,A 82.5656,B 24.8468,C -2.8551,E1 25.0021,E2 0.9891} C_DIS
LIN {X 1.9524,Y 50.5596,Z 66,A 80.5901,B 24.8462,C -2.8609,E1 25.0075,E2 2.9504} C_DIS
LIN {X 4.5473,Y 50.392,Z 66,A 76.9244,B 24.8476,C -2.8485,E1 25.0178,E2 6.6437} C_DIS
LIN {X 7.7154,Y 50.0051,Z 66,A 73.6559,B 24.847,C -2.8536,E1 25.0268,E2 9.8974} C_DIS
LIN {X 10.1647,Y 49.5653,Z 66,A 70.3521,B 24.848,C -2.844,E1 25.0359,E2 13.2201} C_DIS
LIN {X 14.9098,Y 48.3494,Z 66,A 65.3522,B 24.8474,C -2.8501,E1 25.0493,E2 18.1975} C_DIS
LIN {X 17.9346,Y 47.3113,Z 66,A 61.4653,B 24.8482,C -2.8421,E1 25.0595,E2 22.0952} C_DIS
LIN {X 20.2328,Y 46.3753,Z 66,A 58.5677,B 24.8487,C -2.8376,E1 25.067,E2 24.9967} C_DIS
LIN {X 23.127,Y 45.0022,Z 66,A 55.3725,B 24.8484,C -2.841,E1 25.075,E2 28.1752} C_DIS
LIN {X 25.3533,Y 43.7867,Z 66,A 52.5155,B 24.8488,C -2.8374,E1 25.0819,E2 31.0324} C_DIS
LIN {X 27.3866,Y 42.5443,Z 66,A 49.7755,B 24.8493,C -2.8325,E1 25.0884,E2 33.775} C_DIS
LIN {X 29.7154,Y 40.9521,Z 66,A 46.2758,B 24.8504,C -2.8216,E1 25.0964,E2 37.2886} C_DIS
LIN {X 32.327,Y 38.9231,Z 66,A 42.803,B 24.8506,C -2.8199,E1 25.1039,E2 40.7523} C_DIS
LIN {X 34.2545,Y 37.238,Z 66,A 40.1249,B 24.8508,C -2.8185,E1 25.1095,E2 43.4231} C_DIS
LIN {X 35.9197,Y 35.6346,Z 66,A 37.3141,B 24.8517,C -2.8094,E1 25.1151,E2 46.2436} C_DIS
LIN {X 37.5216,Y 33.9443,Z 66,A 34.6938,B 24.8523,C -2.804,E1 25.1201,E2 48.8653} C_DIS
LIN {X 39.3395,Y 31.819,Z 66,A 31.6426,B 24.8528,C -2.799,E1 25.1255,E2 51.9143} C_DIS
LIN {X 41.1079,Y 29.4987,Z 66,A 28.5943,B 24.8531,C -2.7961,E1 25.1306,E2 54.9549} C_DIS
LIN {X 41.9821,Y 28.2413,Z 66,A 26.5805,B 24.8542,C -2.7862,E1 25.1338,E2 56.9819} C_DIS
LIN {X 43.4395,Y 25.9439,Z 66,A 23.6782,B 24.8546,C -2.7819,E1 25.1381,E2 59.8799} C_DIS
LIN {X 44.8259,Y 23.4663,Z 66,A 19.9849,B 24.8565,C -2.7638,E1 25.143,E2 63.5965} C_DIS
LIN {X 46.4863,Y 19.9768,Z 66,A 15.5598,B 24.8579,C -2.7507,E1 25.1481,E2 68.0287} C_DIS
LIN {X 47.5104,Y 17.4013,Z 66,A 12.6775,B 24.8583,C -2.7468,E1 25.1509,E2 70.9042} C_DIS
LIN {X 48.4885,Y 14.4531,Z 66,A 9.4366,B 24.8588,C -2.742,E1 25.1536,E2 74.1379} C_DIS
LIN {X 49.107,Y 12.1885,Z 66,A 6.9418,B 24.8593,C -2.7374,E1 25.1554,E2 76.6293} C_DIS
LIN {X 49.5136,Y 10.4128,Z 66,A 4.5116,B 24.8607,C -2.7237,E1 25.1569,E2 79.0777} C_DIS
LIN {X 50.1014,Y 7.0634,Z 66,A 1.1998,B 24.8607,C -2.7228,E1 25.1584,E2 82.3722} C_DIS
LIN {X 50.4122,Y 4.3201,Z 66,A -2.062,B 24.862,C -2.7103,E1 25.1593,E2 85.6442} C_DIS
LIN {X 50.5784,Y 1.3597,Z 66,A -5.682,B 24.8637,C -2.6945,E1 25.1598,E2 89.2802} C_DIS
LIN {X 50.5839,Y -1.1142,Z 66,A -8.5852,B 24.8648,C -2.6836,E1 25.1597,E2 92.1918} C_DIS
LIN {X 50.4094,Y -4.3514,Z 66,A -12.2203,B 24.8659,C -2.6727,E1 25.1589,E2 95.8311} C_DIS
LIN {X 49.9686,Y -7.95,Z 66,A -15.6951,B 24.8659,C -2.6727,E1 25.1577,E2 99.2855} C_DIS
LIN {X 49.67,Y -9.6399,Z 66,A -17.9364,B 24.8671,C -2.6605,E1 25.1565,E2 101.5424} C_DIS
LIN {X 49.198,Y -11.8149,Z 66,A -20.3426,B 24.8676,C -2.655,E1 25.155,E2 103.9478} C_DIS
LIN {X 48.723,Y -13.6426,Z 66,A -23.1308,B 24.8696,C -2.6352,E1 25.1529,E2 106.7668} C_DIS
LIN {X 47.3113,Y -17.935,Z 66,A -27.5348,B 24.8697,C -2.6341,E1 25.1489,E2 111.1486} C_DIS
LIN {X 46.2717,Y -20.4687,Z 66,A -31.03,B 24.8714,C -2.6168,E1 25.1451,E2 114.6654} C_DIS
LIN {X 45.2005,Y -22.7363,Z 66,A -33.4693,B 24.8714,C -2.6166,E1 25.1421,E2 117.0922} C_DIS
LIN {X 44.4005,Y -24.2622,Z 66,A -35.8389,B 24.8728,C -2.6026,E1 25.1389,E2 119.4826} C_DIS
LIN {X 42.2729,Y -27.8037,Z 66,A -39.776,B 24.8726,C -2.6044,E1 25.1332,E2 123.3953} C_DIS
LIN {X 40.8587,Y -29.8431,Z 66,A -43.5834,B 24.8753,C -2.5769,E1 25.127,E2 127.2492} C_DIS
LIN {X 38.536,Y -32.7874,Z 66,A -46.8628,B 24.8745,C -2.5852,E1 25.1213,E2 130.4939} C_DIS
LIN {X 36.3705,Y -35.1744,Z 66,A -50.862,B 24.8761,C -2.5692,E1 25.1136,E2 134.5132} C_DIS
LIN {X 34.1257,Y -37.3562,Z 66,A -54.9371,B 24.8779,C -2.5507,E1 25.1053,E2 138.6155} C_DIS
LIN {X 31.3117,Y -39.7444,Z 66,A -58.3509,B 24.8773,C -2.5565,E1 25.098,E2 142.0027} C_DIS
LIN {X 28.8012,Y -41.599,Z 66,A -62.2591,B 24.8787,C -2.5421,E1 25.0891,E2 145.9312} C_DIS
LIN {X 26.3707,Y -43.1813,Z 66,A -65.3687,B 24.879,C -2.5393,E1 25.0817,E2 149.0375} C_DIS
LIN {X 23.6059,Y -44.7526,Z 66,A -68.6182,B 24.879,C -2.5398,E1 25.0738,E2 152.2762} C_DIS
LIN {X 21.9837,Y -45.5715,Z 66,A -70.8035,B 24.8795,C -2.5341,E1 25.0683,E2 154.4693} C_DIS
LIN {X 19.6877,Y -46.6094,Z 66,A -74.0644,B 24.8806,C -2.5222,E1 25.06,E2 157.7503} C_DIS
LIN {X 17.2006,Y -47.5834,Z 66,A -77.4324,B 24.8816,C -2.512,E1 25.0511,E2 161.1356} C_DIS
LIN {X 12.7598,Y -48.9615,Z 66,A -81.8538,B 24.8806,C -2.5216,E1 25.0393,E2 165.5265} C_DIS
LIN {X 11.0076,Y -49.3849,Z 66,A -83.9753,B 24.881,C -2.5182,E1 25.0335,E2 167.6531} C_DIS
LIN {X 8.9658,Y -49.7959,Z 66,A -86.5112,B 24.8814,C -2.5131,E1 25.0266,E2 170.1982} C_DIS
LIN {X 6.8955,Y -50.1248,Z 66,A -89.2028,B 24.8821,C -2.5058,E1 25.0191,E2 172.9047} C_DIS
LIN {X 3.368,Y -50.4846,Z 66,A -93.0641,B 24.8821,C -2.5066,E1 25.0083,E2 176.7621} C_DIS
LIN {X 0.2503,Y -50.5897,Z 66,A -95.1216,B 24.8797,C -2.5317,E1 25.0028,E2 178.7595} C_DIS
Enddeposition()
LIN {X 0.2503,Y -50.5897,Z 66,A -95.1216,B 24.8797,C -2.5317,E1 25.0028,E2 178.7595} C_DIS
Startdeposition()
$VEL.CP = VEL_PRINT
LIN {X 1.1982,Y -49.6229,Z 66,A -93.5612,B 24.8773,C -2.5566,E1 25.0073,E2 177.1402} C_DIS
LIN {X 4.4605,Y -49.4368,Z 66,A -90.0326,B 24.8775,C -2.554,E1 25.0171,E2 173.6195} C_DIS
LIN {X 6.6764,Y -49.1871,Z 66,A -87.8811,B 24.8781,C -2.548,E1 25.023,E2 171.4839} C_DIS
LIN {X 8.771,Y -48.8567,Z 66,A -85.0289,B 24.8772,C -2.5572,E1 25.0309,E2 168.613} C_DIS
LIN {X 11.2015,Y -48.3574,Z 66,A -82.5069,B 24.8776,C -2.5535,E1 25.0378,E2 166.103} C_DIS
LIN {X 14.5872,Y -47.4459,Z 66,A -77.3853,B 24.8752,C -2.5778,E1 25.0516,E2 160.9324} C_DIS
LIN {X 19.9865,Y -45.4359,Z 66,A -70.9315,B 24.8747,C -2.5833,E1 25.0683,E2 154.4803} C_DIS
LIN {X 23.0362,Y -43.9686,Z 66,A -67.9109,B 24.8757,C -2.5727,E1 25.0758,E2 151.4929} C_DIS
LIN {X 25.3558,Y -42.6733,Z 66,A -64.41,B 24.8744,C -2.5864,E1 25.0843,E2 147.97} C_DIS
LIN {X 27.6346,Y -41.2345,Z 66,A -61.705,B 24.8746,C -2.5845,E1 25.0906,E2 145.2784} C_DIS
LIN {X 29.4814,Y -39.9345,Z 66,A -58.8608,B 24.8736,C -2.5944,E1 25.0971,E2 142.4208} C_DIS
LIN {X 31.1216,Y -38.6702,Z 66,A -55.8405,B 24.8719,C -2.6119,E1 25.1037,E2 139.3705} C_DIS
LIN {X 34.8126,Y -35.3837,Z 66,A -51.3284,B 24.8729,C -2.6015,E1 25.1129,E2 134.9014} C_DIS
LIN {X 36.6422,Y -33.4854,Z 66,A -47.442,B 24.8706,C -2.6256,E1 25.1204,E2 130.9747} C_DIS
LIN {X 38.2861,Y -31.5929,Z 66,A -44.6184,B 24.87,C -2.6316,E1 25.1254,E2 128.1499} C_DIS
LIN {X 40.2807,Y -29.0062,Z 66,A -41.4602,B 24.8702,C -2.6294,E1 25.1307,E2 125.0121} C_DIS
LIN {X 41.3539,Y -27.4552,Z 66,A -38.8536,B 24.8687,C -2.644,E1 25.1348,E2 122.384} C_DIS
LIN {X 43.1775,Y -24.4868,Z 66,A -35.3241,B 24.8686,C -2.6454,E1 25.1398,E2 118.8692} C_DIS
LIN {X 44.0032,Y -22.97,Z 66,A -32.4856,B 24.8663,C -2.6683,E1 25.1435,E2 115.9915} C_DIS
LIN {X 46.1878,Y -18.1823,Z 66,A -26.2022,B 24.864,C -2.6906,E1 25.1504,E2 109.6897} C_DIS
LIN {X 47.9201,Y -12.9452,Z 66,A -20.928,B 24.8643,C -2.6877,E1 25.1547,E2 104.4523} C_DIS
LIN {X 48.4357,Y -10.8575,Z 66,A -18.2984,B 24.8633,C -2.6985,E1 25.1564,E2 101.8126} C_DIS
LIN {X 48.9356,Y -8.3207,Z 66,A -15.3056,B 24.8623,C -2.708,E1 25.1579,E2 98.8149} C_DIS
LIN {X 49.3328,Y -5.4935,Z 66,A -12.0267,B 24.8613,C -2.718,E1 25.159,E2 95.5315} C_DIS
LIN {X 49.5844,Y -2.2906,Z 66,A -7.8333,B 24.859,C -2.7397,E1 25.1597,E2 91.3118} C_DIS
LIN {X 49.6203,Y 1.3142,Z 66,A -3.8823,B 24.8581,C -2.7484,E1 25.1597,E2 87.3637} C_DIS
LIN {X 49.4309,Y 4.5276,Z 66,A -0.3043,B 24.8572,C -2.7572,E1 25.1588,E2 83.7862} C_DIS
LIN {X 48.9231,Y 8.3934,Z 66,A 3.8961,B 24.8564,C -2.7649,E1 25.1571,E2 79.5922} C_DIS
LIN {X 48.431,Y 10.879,Z 66,A 6.7484,B 24.8556,C -2.7723,E1 25.1555,E2 76.7391} C_DIS
LIN {X 47.943,Y 12.8601,Z 66,A 8.9406,B 24.8552,C -2.7761,E1 25.154,E2 74.5506} C_DIS
LIN {X 47.2387,Y 15.2448,Z 66,A 12.3137,B 24.8533,C -2.7947,E1 25.1511,E2 71.1527} C_DIS
LIN {X 46.1126,Y 18.371,Z 66,A 15.8836,B 24.8527,C -2.8003,E1 25.1476,E2 67.5893} C_DIS
LIN {X 44.9575,Y 21.0416,Z 66,A 18.7352,B 24.8527,C -2.7995,E1 25.1444,E2 64.755} C_DIS
LIN {X 43.2501,Y 24.3592,Z 66,A 23.6309,B 24.8503,C -2.8228,E1 25.138,E2 59.8301} C_DIS
LIN {X 41.8436,Y 26.7027,Z 66,A 26.4143,B 24.8503,C -2.8235,E1 25.1339,E2 57.0591} C_DIS
LIN {X 40.4374,Y 28.7877,Z 66,A 29.7385,B 24.8486,C -2.839,E1 25.1286,E2 53.7146} C_DIS
LIN {X 38.8024,Y 30.9568,Z 66,A 32.7717,B 24.848,C -2.8443,E1 25.1234,E2 50.6831} C_DIS
LIN {X 36.8381,Y 33.2701,Z 66,A 35.7275,B 24.8483,C -2.8415,E1 25.118,E2 47.7471} C_DIS
LIN {X 35.8939,Y 34.2863,Z 66,A 37.5742,B 24.8474,C -2.8497,E1 25.1144,E2 45.8891} C_DIS
LIN {X 34.3325,Y 35.8499,Z 66,A 40.1824,B 24.8467,C -2.8561,E1 25.1092,E2 43.2767} C_DIS
LIN {X 32.3941,Y 37.6102,Z 66,A 43.0448,B 24.8464,C -2.8589,E1 25.1032,E2 40.4191} C_DIS
LIN {X 30.5641,Y 39.1128,Z 66,A 46.0398,B 24.8454,C -2.8687,E1 25.0967,E2 37.4119} C_DIS
LIN {X 28.2888,Y 40.788,Z 66,A 49.3904,B 24.8446,C -2.8759,E1 25.089,E2 34.0562} C_DIS
LIN {X 25.6862,Y 42.4752,Z 66,A 52.5605,B 24.8449,C -2.8736,E1 25.0816,E2 30.9016} C_DIS
LIN {X 23.9991,Y 43.4509,Z 66,A 54.798,B 24.8445,C -2.8765,E1 25.0762,E2 28.6638} C_DIS
LIN {X 22.4074,Y 44.2924,Z 66,A 57.3539,B 24.8433,C -2.8879,E1 25.0698,E2 26.088} C_DIS
LIN {X 19.6113,Y 45.5993,Z 66,A 60.339,B 24.844,C -2.8813,E1 25.0622,E2 23.1259} C_DIS
LIN {X 17.3768,Y 46.4966,Z 66,A 63.6967,B 24.8426,C -2.8944,E1 25.0534,E2 19.7444} C_DIS
LIN {X 14.5213,Y 47.466,Z 66,A 67.5362,B 24.8416,C -2.9035,E1 25.0431,E2 15.8904} C_DIS
LIN {X 9.9647,Y 48.6273,Z 66,A 72.176,B 24.8428,C -2.8924,E1 25.0306,E2 11.2835} C_DIS
LIN {X 7.7226,Y 49.0336,Z 66,A 74.713,B 24.8428,C -2.8916,E1 25.0237,E2 8.7509} C_DIS
LIN {X 4.7904,Y 49.4062,Z 66,A 78.7103,B 24.8417,C -2.9023,E1 25.0125,E2 4.7312} C_DIS
LIN {X 2.0167,Y 49.5969,Z 66,A 81.3279,B 24.8428,C -2.8921,E1 25.0053,E2 2.1387} C_DIS
LIN {X -0.5634,Y 49.6346,Z 66,A 84.3677,B 24.8428,C -2.8926,E1 24.9968,E2 -0.9021} C_DIS
LIN {X -2.9898,Y 49.5475,Z 66,A 87.9531,B 24.8415,C -2.9047,E1 24.9867,E2 -4.5173} C_DIS
LIN {X -5.6427,Y 49.3162,Z 66,A 90.8446,B 24.842,C -2.9,E1 24.9787,E2 -7.3993} C_DIS
LIN {X -8.8996,Y 48.8336,Z 66,A 94.1771,B 24.8431,C -2.8897,E1 24.9696,E2 -10.7104} C_DIS
LIN {X -11.1143,Y 48.3774,Z 66,A 96.7592,B 24.8434,C -2.887,E1 24.9625,E2 -13.2892} C_DIS
LIN {X -13.544,Y 47.7542,Z 66,A 99.3745,B 24.8442,C -2.8796,E1 24.9555,E2 -15.891} C_DIS
LIN {X -15.7349,Y 47.0775,Z 66,A 102.6265,B 24.8435,C -2.8862,E1 24.9468,E2 -19.1645} C_DIS
LIN {X -18.8942,Y 45.9011,Z 66,A 106.1691,B 24.8446,C -2.8755,E1 24.9377,E2 -22.6893} C_DIS
LIN {X -20.8562,Y 45.0436,Z 66,A 108.9627,B 24.8445,C -2.8769,E1 24.9305,E2 -25.493} C_DIS
LIN {X -23.6486,Y 43.6423,Z 66,A 112.8208,B 24.8447,C -2.8749,E1 24.921,E2 -29.357} C_DIS
LIN {X -27.4333,Y 41.3678,Z 66,A 117.1671,B 24.8469,C -2.8542,E1 24.9107,E2 -33.6675} C_DIS
LIN {X -29.1651,Y 40.1651,Z 66,A 120.3257,B 24.8463,C -2.8603,E1 24.9035,E2 -36.8516} C_DIS
LIN {X -32.1239,Y 37.8414,Z 66,A 124.3999,B 24.8477,C -2.847,E1 24.8947,E2 -40.9094} C_DIS
LIN {X -34.3259,Y 35.8557,Z 66,A 127.579,B 24.8489,C -2.8356,E1 24.8882,E2 -44.0742} C_DIS
LIN {X -35.804,Y 34.3801,Z 66,A 130.0226,B 24.8495,C -2.8304,E1 24.8835,E2 -46.5157} C_DIS
LIN {X -37.122,Y 32.9529,Z 66,A 132.6708,B 24.8495,C -2.8307,E1 24.8785,E2 -49.1766} C_DIS
LIN {X -39.1494,Y 30.5174,Z 66,A 136.6488,B 24.85,C -2.8259,E1 24.8716,E2 -53.1618} C_DIS
LIN {X -41.897,Y 26.6192,Z 66,A 141.1716,B 24.853,C -2.797,E1 24.8645,E2 -57.6378} C_DIS
LIN {X -43.5131,Y 23.8851,Z 66,A 145.9551,B 24.8525,C -2.8025,E1 24.8578,E2 -62.4594} C_DIS
LIN {X -45.0608,Y 20.8188,Z 66,A 149.2597,B 24.8547,C -2.7816,E1 24.8538,E2 -65.7319} C_DIS
LIN {X -46.0851,Y 18.4408,Z 66,A 152.559,B 24.8551,C -2.777,E1 24.8503,E2 -69.0387} C_DIS
LIN {X -46.8604,Y 16.3712,Z 66,A 155.303,B 24.8557,C -2.772,E1 24.8478,E2 -71.7863} C_DIS
LIN {X -47.964,Y 12.7825,Z 66,A 159.0081,B 24.858,C -2.7499,E1 24.8449,E2 -75.4599} C_DIS
LIN {X -48.3276,Y 11.3277,Z 66,A 161.0711,B 24.858,C -2.7492,E1 24.8435,E2 -77.5332} C_DIS
LIN {X -48.8743,Y 8.6727,Z 66,A 163.9337,B 24.8594,C -2.7357,E1 24.842,E2 -80.3805} C_DIS
LIN {X -49.1566,Y 6.8924,Z 66,A 166.7304,B 24.8591,C -2.7392,E1 24.8409,E2 -83.2022} C_DIS
LIN {X -49.4846,Y 3.8965,Z 66,A 170.1894,B 24.8602,C -2.7279,E1 24.8401,E2 -86.655} C_DIS
LIN {X -49.6358,Y 0.3564,Z 66,A 173.7898,B 24.8623,C -2.7082,E1 24.8398,E2 -90.2301} C_DIS
LIN {X -49.5962,Y -2.0123,Z 66,A 177.0126,B 24.8624,C -2.7065,E1 24.8401,E2 -93.4681} C_DIS
LIN {X -49.4115,Y -4.7373,Z 66,A 179.8789,B 24.8638,C -2.6927,E1 24.8407,E2 -96.3185} C_DIS
LIN {X -48.9333,Y -8.3347,Z 66,A -175.5527,B 24.8646,C -2.6851,E1 24.8426,E2 -100.896} C_DIS
LIN {X -48.4618,Y -10.7421,Z 66,A -172.6227,B 24.8653,C -2.6779,E1 24.8444,E2 -103.8261} C_DIS
LIN {X -47.4627,Y -14.5333,Z 66,A -168.6082,B 24.8674,C -2.6573,E1 24.8474,E2 -107.8144} C_DIS
LIN {X -46.6918,Y -16.8467,Z 66,A -165.9784,B 24.8685,C -2.6465,E1 24.8498,E2 -110.4334} C_DIS
LIN {X -46.1467,Y -18.2868,Z 66,A -164.1677,B 24.8689,C -2.6419,E1 24.8516,E2 -112.2433} C_DIS
LIN {X -45.5525,Y -19.7203,Z 66,A -162.1496,B 24.8691,C -2.6401,E1 24.8538,E2 -114.2683} C_DIS
LIN {X -44.5921,Y -21.8049,Z 66,A -159.4109,B 24.8697,C -2.6341,E1 24.8571,E2 -117.0075} C_DIS
LIN {X -43.2856,Y -24.2957,Z 66,A -156.3808,B 24.8709,C -2.6223,E1 24.8611,E2 -120.0256} C_DIS
LIN {X -42.0014,Y -26.4529,Z 66,A -152.8184,B 24.8707,C -2.6247,E1 24.8664,E2 -123.6117} C_DIS
LIN {X -40.6931,Y -28.4252,Z 66,A -149.7707,B 24.8709,C -2.6226,E1 24.8713,E2 -126.6696} C_DIS
LIN {X -38.5726,Y -31.242,Z 66,A -145.5794,B 24.8716,C -2.615,E1 24.8786,E2 -130.8624} C_DIS
LIN {X -36.3752,Y -33.7759,Z 66,A -141.4304,B 24.872,C -2.6109,E1 24.8865,E2 -135.0197} C_DIS
LIN {X -34.092,Y -36.0785,Z 66,A -139.2693,B 24.8751,C -2.5791,E1 24.8906,E2 -137.1141} C_DIS
LIN {X -32.8339,Y -37.2268,Z 66,A -136.2231,B 24.8739,C -2.5919,E1 24.8971,E2 -140.2027} C_DIS
LIN {X -29.9232,Y -39.6043,Z 66,A -132.5426,B 24.8756,C -2.574,E1 24.9051,E2 -143.8542} C_DIS
LIN {X -28.1132,Y -40.91,Z 66,A -130.1216,B 24.8763,C -2.5674,E1 24.9106,E2 -146.2678} C_DIS
LIN {X -26.8508,Y -41.7486,Z 66,A -128.2083,B 24.8763,C -2.5673,E1 24.9151,E2 -148.187} C_DIS
LIN {X -24.9951,Y -42.8855,Z 66,A -125.2985,B 24.876,C -2.57,E1 24.9221,E2 -151.1123} C_DIS
LIN {X -21.6708,Y -44.6577,Z 66,A -121.0458,B 24.8767,C -2.5631,E1 24.9327,E2 -155.36} C_DIS
LIN {X -18.6576,Y -45.9979,Z 66,A -117.3954,B 24.8773,C -2.5567,E1 24.942,E2 -159.0035} C_DIS
LIN {X -15.1197,Y -47.2786,Z 66,A -112.5543,B 24.8768,C -2.5614,E1 24.9549,E2 -163.8651} C_DIS
LIN {X -11.8843,Y -48.1931,Z 66,A -108.9973,B 24.8776,C -2.5537,E1 24.9644,E2 -167.4091} C_DIS
LIN {X -8.6682,Y -48.8751,Z 66,A -105.3011,B 24.8779,C -2.5506,E1 24.9746,E2 -171.1019} C_DIS
LIN {X -6.5081,Y -49.2094,Z 66,A -103.0684,B 24.8784,C -2.5451,E1 24.9807,E2 -173.3234} C_DIS
LIN {X -4.9258,Y -49.3929,Z 66,A -101.3207,B 24.8786,C -2.5433,E1 24.9855,E2 -175.068} C_DIS
LIN {X -2.8889,Y -49.5537,Z 66,A -98.4206,B 24.8777,C -2.5528,E1 24.9937,E2 -177.9914} C_DIS
LIN {X 0.2503,Y -49.6229,Z 66,A -96.0036,B 24.8796,C -2.5326,E1 25.0003,E2 -180.3608} C_DIS
Enddeposition()
LIN {X 0.2503,Y -49.6229,Z 66,A -96.0036,B 24.8796,C -2.5326,E1 25.0003,E2 -180.3608} C_DIS
Startdeposition()
$VEL.CP = VEL_PRINT
LIN {X -0.1432,Y -48.6788,Z 66,A -96.9562,B 24.8788,C -2.5407,E1 24.9977,E2 -179.4275} C_DIS
LIN {X -2.4572,Y -48.6166,Z 66,A -99.8534,B 24.8791,C -2.5376,E1 24.9896,E2 -176.5222} C_DIS
LIN {X -5.8919,Y -48.321,Z 66,A -103.6829,B 24.8787,C -2.5417,E1 24.979,E2 -172.7003} C_DIS
LIN {X -8.3096,Y -47.9648,Z 66,A -106.5639,B 24.8787,C -2.5424,E1 24.971,E2 -169.8184} C_DIS
LIN {X -10.3433,Y -47.5671,Z 66,A -108.8696,B 24.8784,C -2.5456,E1 24.9647,E2 -167.5175} C_DIS
LIN {X -12.0717,Y -47.1582,Z 66,A -110.8434,B 24.8781,C -2.5486,E1 24.9594,E2 -165.5481} C_DIS
LIN {X -14.1303,Y -46.5827,Z 66,A -113.7138,B 24.8784,C -2.5446,E1 24.9517,E2 -162.6635} C_DIS
LIN {X -17.4057,Y -45.4606,Z 66,A -117.9414,B 24.8784,C -2.5457,E1 24.9405,E2 -158.4301} C_DIS
LIN {X -19.9304,Y -44.4117,Z 66,A -120.8777,B 24.8776,C -2.5534,E1 24.933,E2 -155.5052} C_DIS
LIN {X -22.0181,Y -43.4144,Z 66,A -123.5366,B 24.8772,C -2.5576,E1 24.9264,E2 -152.8494} C_DIS
LIN {X -23.6568,Y -42.5439,Z 66,A -125.584,B 24.8767,C -2.5625,E1 24.9214,E2 -150.8079} C_DIS
LIN {X -25.4444,Y -41.4998,Z 66,A -128.4188,B 24.877,C -2.56,E1 24.9145,E2 -147.9584} C_DIS
LIN {X -27.4174,Y -40.2235,Z 66,A -131.1893,B 24.8766,C -2.5642,E1 24.9081,E2 -145.1888} C_DIS
LIN {X -30.2926,Y -38.105,Z 66,A -135.6235,B 24.8762,C -2.5681,E1 24.8983,E2 -140.7479} C_DIS
LIN {X -33.2037,Y -35.5973,Z 66,A -141.1505,B 24.8767,C -2.5626,E1 24.8868,E2 -135.1855} C_DIS
LIN {X -35.6897,Y -33.1046,Z 66,A -143.5815,B 24.8735,C -2.5956,E1 24.8822,E2 -132.8229} C_DIS
LIN {X -37.6319,Y -30.8779,Z 66,A -147.169,B 24.8729,C -2.6018,E1 24.8757,E2 -129.2339} C_DIS
LIN {X -39.8535,Y -27.9527,Z 66,A -151.4243,B 24.8718,C -2.6131,E1 24.8685,E2 -124.9851} C_DIS
LIN {X -41.7946,Y -24.9566,Z 66,A -155.9377,B 24.8712,C -2.6194,E1 24.8618,E2 -120.4638} C_DIS
LIN {X -43.1595,Y -22.5139,Z 66,A -159.6058,B 24.8708,C -2.623,E1 24.8568,E2 -116.785} C_DIS
LIN {X -44.2526,Y -20.2809,Z 66,A -162.1811,B 24.8696,C -2.6358,E1 24.8538,E2 -114.2263} C_DIS
LIN {X -45.4035,Y -17.5536,Z 66,A -165.407,B 24.8682,C -2.6491,E1 24.8504,E2 -111.0144} C_DIS
LIN {X -46.204,Y -15.3231,Z 66,A -168.8819,B 24.8683,C -2.648,E1 24.8472,E2 -107.5169} C_DIS
LIN {X -47.0104,Y -12.6349,Z 66,A -172.0519,B 24.8672,C -2.6595,E1 24.8447,E2 -104.3562} C_DIS
LIN {X -47.5847,Y -10.2621,Z 66,A -174.4907,B 24.8657,C -2.674,E1 24.8432,E2 -101.9377} C_DIS
LIN {X -47.8972,Y -8.6877,Z 66,A -176.6392,B 24.8655,C -2.6763,E1 24.8421,E2 -99.7819} C_DIS
LIN {X -48.2144,Y -6.7084,Z 66,A -179.4152,B 24.8653,C -2.678,E1 24.841,E2 -96.9935} C_DIS
LIN {X -48.4911,Y -4.2699,Z 66,A 178.0682,B 24.8639,C -2.6919,E1 24.8403,E2 -94.495} C_DIS
LIN {X -48.6546,Y -1.5292,Z 66,A 174.4366,B 24.8634,C -2.6967,E1 24.8398,E2 -90.8532} C_DIS
LIN {X -48.6585,Y 1.3981,Z 66,A 171.0583,B 24.8622,C -2.7084,E1 24.8399,E2 -87.4826} C_DIS
LIN {X -48.4694,Y 4.5101,Z 66,A 166.9436,B 24.8616,C -2.7142,E1 24.8408,E2 -83.3568} C_DIS
LIN {X -47.9338,Y 8.4836,Z 66,A 162.9068,B 24.8592,C -2.7379,E1 24.8425,E2 -79.3528} C_DIS
LIN {X -47.5381,Y 10.4761,Z 66,A 160.4018,B 24.8586,C -2.7439,E1 24.844,E2 -76.8472} C_DIS
LIN {X -47.0218,Y 12.593,Z 66,A 157.4665,B 24.8583,C -2.7469,E1 24.846,E2 -73.9021} C_DIS
LIN {X -45.9309,Y 16.1237,Z 66,A 153.8207,B 24.8559,C -2.7695,E1 24.8491,E2 -70.2895} C_DIS
LIN {X -45.2403,Y 17.9695,Z 66,A 151.1478,B 24.8557,C -2.7718,E1 24.8518,E2 -67.607} C_DIS
LIN {X -44.3832,Y 19.9931,Z 66,A 148.4557,B 24.855,C -2.778,E1 24.8548,E2 -64.9149} C_DIS
LIN {X -43.0986,Y 22.6301,Z 66,A 144.7175,B 24.8544,C -2.7842,E1 24.8595,E2 -61.1714} C_DIS
LIN {X -41.8766,Y 24.8187,Z 66,A 141.8676,B 24.8534,C -2.7938,E1 24.8635,E2 -58.3298} C_DIS
LIN {X -40.8704,Y 26.4431,Z 66,A 139.1292,B 24.8534,C -2.7934,E1 24.8676,E2 -55.5766} C_DIS
LIN {X -38.454,Y 29.8486,Z 66,A 134.3079,B 24.8519,C -2.8077,E1 24.8757,E2 -50.7661} C_DIS
LIN {X -35.5775,Y 33.2236,Z 66,A 129.9016,B 24.8493,C -2.8319,E1 24.8837,E2 -46.3977} C_DIS
LIN {X -34.603,Y 34.238,Z 66,A 127.2207,B 24.8504,C -2.8216,E1 24.889,E2 -43.6809} C_DIS
LIN {X -31.448,Y 37.1574,Z 66,A 122.2359,B 24.8491,C -2.8339,E1 24.8994,E2 -38.7058} C_DIS
LIN {X -27.6764,Y 40.0456,Z 66,A 117.423,B 24.8467,C -2.8563,E1 24.9101,E2 -33.9292} C_DIS
LIN {X -24.9103,Y 41.8223,Z 66,A 112.7165,B 24.8473,C -2.8513,E1 24.9214,E2 -29.196} C_DIS
LIN {X -22.045,Y 43.4009,Z 66,A 109.4825,B 24.8456,C -2.8666,E1 24.9293,E2 -25.9895} C_DIS
LIN {X -19.6953,Y 44.5164,Z 66,A 106.121,B 24.8456,C -2.8666,E1 24.9378,E2 -22.62} C_DIS
LIN {X -17.3546,Y 45.4796,Z 66,A 103.2256,B 24.845,C -2.8719,E1 24.9453,E2 -19.7308} C_DIS
LIN {X -14.159,Y 46.574,Z 66,A 99.1377,B 24.8447,C -2.8748,E1 24.9562,E2 -15.6424} C_DIS
LIN {X -11.3192,Y 47.3444,Z 66,A 95.5604,B 24.8445,C -2.8764,E1 24.9659,E2 -12.0637} C_DIS
LIN {X -8.0695,Y 48.0052,Z 66,A 91.871,B 24.8439,C -2.8827,E1 24.976,E2 -8.3854} C_DIS
LIN {X -5.401,Y 48.3782,Z 66,A 88.7163,B 24.8436,C -2.8848,E1 24.9847,E2 -5.2335} C_DIS
LIN {X -2.671,Y 48.6054,Z 66,A 85.5293,B 24.8434,C -2.8867,E1 24.9936,E2 -2.0498} C_DIS
LIN {X -0.5061,Y 48.676,Z 66,A 82.8957,B 24.8435,C -2.886,E1 25.0009,E2 0.5856} C_DIS
LIN {X 2.1109,Y 48.6328,Z 66,A 80.1291,B 24.8429,C -2.8914,E1 25.0086,E2 3.3387} C_DIS
LIN {X 4.5469,Y 48.466,Z 66,A 76.9331,B 24.8435,C -2.886,E1 25.0175,E2 6.5461} C_DIS
LIN {X 7.2513,Y 48.1357,Z 66,A 73.7545,B 24.8435,C -2.8857,E1 25.0263,E2 9.7226} C_DIS
LIN {X 9.7647,Y 47.6893,Z 66,A 70.8414,B 24.8435,C -2.886,E1 25.0343,E2 12.6315} C_DIS
LIN {X 12.1446,Y 47.1389,Z 66,A 67.3422,B 24.8448,C -2.8739,E1 25.0439,E2 16.1543} C_DIS
LIN {X 15.4123,Y 46.1747,Z 66,A 64.3768,B 24.8432,C -2.8887,E1 25.0517,E2 19.0793} C_DIS
LIN {X 17.0911,Y 45.5797,Z 66,A 61.9436,B 24.844,C -2.881,E1 25.0581,E2 21.5256} C_DIS
LIN {X 19.5115,Y 44.5971,Z 66,A 59.1484,B 24.8439,C -2.8827,E1 25.0652,E2 24.3102} C_DIS
LIN {X 21.6865,Y 43.5811,Z 66,A 56.0386,B 24.8448,C -2.8744,E1 25.0731,E2 27.4317} C_DIS
LIN {X 23.7917,Y 42.4686,Z 66,A 53.1477,B 24.8453,C -2.8691,E1 25.0802,E2 30.3268} C_DIS
LIN {X 25.9182,Y 41.2055,Z 66,A 50.361,B 24.8456,C -2.867,E1 25.0868,E2 33.1097} C_DIS
LIN {X 28.079,Y 39.7649,Z 66,A 46.76,B 24.8471,C -2.8523,E1 25.0952,E2 36.7333} C_DIS
LIN {X 30.9548,Y 37.5694,Z 66,A 43.4217,B 24.8462,C -2.8614,E1 25.1024,E2 40.0376} C_DIS
LIN {X 32.5823,Y 36.1666,Z 66,A 40.3864,B 24.8477,C -2.8473,E1 25.1088,E2 43.0945} C_DIS
LIN {X 34.2561,Y 34.5853,Z 66,A 37.9983,B 24.8477,C -2.8477,E1 25.1136,E2 45.4716} C_DIS
LIN {X 35.5293,Y 33.276,Z 66,A 35.8524,B 24.8481,C -2.8432,E1 25.1177,E2 47.6189} C_DIS
LIN {X 37.2894,Y 31.291,Z 66,A 32.4267,B 24.8495,C -2.8305,E1 25.124,E2 51.0591} C_DIS
LIN {X 38.4968,Y 29.7931,Z 66,A 30.3437,B 24.8497,C -2.8286,E1 25.1276,E2 53.1369} C_DIS
LIN {X 39.9189,Y 27.8586,Z 66,A 27.5171,B 24.8504,C -2.8217,E1 25.1322,E2 55.9661} C_DIS
LIN {X 41.0182,Y 26.2133,Z 66,A 25.4394,B 24.8505,C -2.8206,E1 25.1354,E2 58.036} C_DIS
LIN {X 42.5527,Y 23.641,Z 66,A 20.7981,B 24.8538,C -2.7902,E1 25.1419,E2 62.7253} C_DIS
LIN {X 44.2418,Y 20.3045,Z 66,A 17.1896,B 24.8534,C -2.7932,E1 25.1462,E2 66.3072} C_DIS
LIN {X 45.519,Y 17.2523,Z 66,A 13.8201,B 24.8535,C -2.7923,E1 25.1497,E2 69.6602} C_DIS
LIN {X 46.0377,Y 15.8139,Z 66,A 11.4985,B 24.8551,C -2.777,E1 25.1519,E2 72.0051} C_DIS
LIN {X 46.9331,Y 12.9188,Z 66,A 8.1414,B 24.8558,C -2.7705,E1 25.1546,E2 75.3583} C_DIS
LIN {X 47.7282,Y 9.5728,Z 66,A 4.3522,B 24.8566,C -2.7634,E1 25.1569,E2 79.1425} C_DIS
LIN {X 48.1092,Y 7.4242,Z 66,A 1.4841,B 24.858,C -2.7496,E1 25.1582,E2 82.0263} C_DIS
LIN {X 48.4481,Y 4.7353,Z 66,A -1.4111,B 24.8584,C -2.7455,E1 25.1591,E2 84.9141} C_DIS
LIN {X 48.5988,Y 2.7898,Z 66,A -4.224,B 24.8602,C -2.7282,E1 25.1597,E2 87.7512} C_DIS
LIN {X 48.6767,Y 0.3569,Z 66,A -6.5082,B 24.86,C -2.7306,E1 25.1597,E2 90.0161} C_DIS
LIN {X 48.6242,Y -2.304,Z 66,A -10.1084,B 24.8619,C -2.7115,E1 25.1595,E2 93.64} C_DIS
LIN {X 48.4217,Y -4.9955,Z 66,A -12.9645,B 24.8623,C -2.7078,E1 25.1587,E2 96.4879} C_DIS
LIN {X 48.1503,Y -7.1561,Z 66,A -15.4493,B 24.863,C -2.7013,E1 25.1578,E2 98.9734} C_DIS
LIN {X 47.6468,Y -9.9679,Z 66,A -19.5225,B 24.8654,C -2.6769,E1 25.1556,E2 103.0807} C_DIS
LIN {X 46.9939,Y -12.6961,Z 66,A -22.9438,B 24.8667,C -2.6643,E1 25.1531,E2 106.512} C_DIS
LIN {X 45.4283,Y -17.4894,Z 66,A -27.9151,B 24.8667,C -2.6651,E1 25.1486,E2 111.4535} C_DIS
LIN {X 44.1756,Y -20.4478,Z 66,A -32.3034,B 24.8689,C -2.642,E1 25.1437,E2 115.8723} C_DIS
LIN {X 42.6456,Y -23.4735,Z 66,A -35.934,B 24.8694,C -2.6375,E1 25.1389,E2 119.4946} C_DIS
LIN {X 41.2837,Y -25.7929,Z 66,A -38.9377,B 24.87,C -2.6318,E1 25.1346,E2 122.4965} C_DIS
LIN {X 39.5029,Y -28.4455,Z 66,A -43.2802,B 24.8721,C -2.6104,E1 25.1276,E2 126.8683} C_DIS
LIN {X 37.5946,Y -30.9244,Z 66,A -46.0606,B 24.8713,C -2.6181,E1 25.1228,E2 129.6175} C_DIS
LIN {X 35.5645,Y -33.2377,Z 66,A -50.3891,B 24.8735,C -2.5956,E1 25.1147,E2 133.9799} C_DIS
LIN {X 32.6972,Y -36.0615,Z 66,A -55.3302,B 24.875,C -2.5808,E1 25.1046,E2 138.9357} C_DIS
LIN {X 30.3362,Y -38.0706,Z 66,A -58.1336,B 24.8742,C -2.5887,E1 25.0986,E2 141.7099} C_DIS
LIN {X 27.8365,Y -39.9343,Z 66,A -62.3935,B 24.876,C -2.5703,E1 25.0889,E2 145.9984} C_DIS
LIN {X 25.1464,Y -41.6809,Z 66,A -65.7356,B 24.8759,C -2.5712,E1 25.081,E2 149.3276} C_DIS
LIN {X 22.7882,Y -43.0154,Z 66,A -68.969,B 24.8765,C -2.5649,E1 25.0731,E2 152.5665} C_DIS
LIN {X 19.718,Y -44.5063,Z 66,A -73.4837,B 24.8779,C -2.5499,E1 25.0616,E2 157.1054} C_DIS
LIN {X 16.6758,Y -45.7333,Z 66,A -77.5193,B 24.8787,C -2.5417,E1 25.051,E2 161.1518} C_DIS
LIN {X 11.3587,Y -47.3352,Z 66,A -83.9301,B 24.8792,C -2.537,E1 25.0338,E2 167.5633} C_DIS
LIN {X 7.1966,Y -48.1444,Z 66,A -88.1855,B 24.8783,C -2.5459,E1 25.0222,E2 171.7931} C_DIS
LIN {X 4.9759,Y -48.4233,Z 66,A -90.7524,B 24.8783,C -2.5455,E1 25.015,E2 174.3591} C_DIS
LIN {X 2.9514,Y -48.5899,Z 66,A -93.4543,B 24.879,C -2.5391,E1 25.0075,E2 177.0749} C_DIS
LIN {X 0.2375,Y -48.6736,Z 66,A -95.2944,B 24.8768,C -2.5613,E1 25.0025,E2 178.8619} C_DIS
Enddeposition()
LIN {X 0.2375,Y -48.6736,Z 66,A -95.2944,B 24.8768,C -2.5613,E1 25.0025,E2 178.8619} C_DIS
Startdeposition()
$VEL.CP = VEL_PRINT
LIN {X 0.8365,Y -47.7122,Z 66,A -94.5803,B 24.8752,C -2.5778,E1 25.0046,E2 178.1088} C_DIS
LIN {X 2.7427,Y -47.6409,Z 66,A -92.0711,B 24.8748,C -2.5823,E1 25.0116,E2 175.5895} C_DIS
LIN {X 5.5052,Y -47.4011,Z 66,A -88.6264,B 24.8744,C -2.5861,E1 25.0212,E2 172.138} C_DIS
LIN {X 7.6589,Y -47.1015,Z 66,A -86.4302,B 24.875,C -2.5808,E1 25.0272,E2 169.9566} C_DIS
LIN {X 9.6181,Y -46.7403,Z 66,A -83.5964,B 24.874,C -2.5905,E1 25.035,E2 167.1032} C_DIS
LIN {X 11.5694,Y -46.2959,Z 66,A -81.2975,B 24.874,C -2.591,E1 25.0413,E2 164.8064} C_DIS
LIN {X 14.4925,Y -45.4656,Z 66,A -77.5524,B 24.8734,C -2.5968,E1 25.0513,E2 161.0541} C_DIS
LIN {X 16.8929,Y -44.6296,Z 66,A -74.8123,B 24.8736,C -2.5951,E1 25.0585,E2 158.3236} C_DIS
LIN {X 19.4303,Y -43.5845,Z 66,A -71.1886,B 24.8725,C -2.6059,E1 25.0678,E2 154.6831} C_DIS
LIN {X 22.5274,Y -42.0676,Z 66,A -66.8085,B 24.8714,C -2.617,E1 25.0787,E2 150.2886} C_DIS
LIN {X 24.8856,Y -40.7172,Z 66,A -64.3482,B 24.8723,C -2.6081,E1 25.0846,E2 147.8571} C_DIS
LIN {X 26.5806,Y -39.6317,Z 66,A -61.5985,B 24.8712,C -2.6189,E1 25.091,E2 145.0909} C_DIS
LIN {X 28.489,Y -38.2818,Z 66,A -58.682,B 24.8705,C -2.6267,E1 25.0976,E2 142.1663} C_DIS
LIN {X 31.0963,Y -36.1964,Z 66,A -54.5783,B 24.8694,C -2.6372,E1 25.1065,E2 138.0534} C_DIS
LIN {X 33.4664,Y -34.0173,Z 66,A -50.8129,B 24.8687,C -2.6443,E1 25.1141,E2 134.2867} C_DIS
LIN {X 35.6873,Y -31.6786,Z 66,A -47.4014,B 24.8687,C -2.645,E1 25.1205,E2 130.8885} C_DIS
LIN {X 36.8869,Y -30.2751,Z 66,A -44.7056,B 24.8672,C -2.6598,E1 25.1254,E2 128.1699} C_DIS
LIN {X 38.4732,Y -28.2306,Z 66,A -41.8467,B 24.8668,C -2.6633,E1 25.1302,E2 125.3165} C_DIS
LIN {X 39.9204,Y -26.1448,Z 66,A -39.1215,B 24.8666,C -2.6654,E1 25.1344,E2 122.5999} C_DIS
LIN {X 40.68,Y -24.9455,Z 66,A -36.6867,B 24.8647,C -2.6843,E1 25.138,E2 120.1326} C_DIS
LIN {X 42.5364,Y -21.6292,Z 66,A -32.3537,B 24.8638,C -2.6929,E1 25.1437,E2 115.802} C_DIS
LIN {X 43.9708,Y -18.5396,Z 66,A -28.7043,B 24.8635,C -2.6964,E1 25.1479,E2 112.1642} C_DIS
LIN {X 44.6671,Y -16.7936,Z 66,A -26.0024,B 24.8619,C -2.712,E1 25.1506,E2 109.4406} C_DIS
LIN {X 45.775,Y -13.4824,Z 66,A -22.0127,B 24.861,C -2.7208,E1 25.154,E2 105.4526} C_DIS
LIN {X 46.2873,Y -11.6039,Z 66,A -19.3962,B 24.8597,C -2.7336,E1 25.1558,E2 102.8211} C_DIS
LIN {X 46.9011,Y -8.8014,Z 66,A -16.5587,B 24.8597,C -2.7323,E1 25.1573,E2 100.003} C_DIS
LIN {X 47.2648,Y -6.5743,Z 66,A -13.5513,B 24.8583,C -2.7467,E1 25.1586,E2 96.9793} C_DIS
LIN {X 47.5103,Y -4.4655,Z 66,A -11.4418,B 24.8583,C -2.7461,E1 25.1592,E2 94.8838} C_DIS
LIN {X 47.6492,Y -2.5934,Z 66,A -8.975,B 24.8572,C -2.7574,E1 25.1596,E2 92.4049} C_DIS
LIN {X 47.7173,Y -0.4815,Z 66,A -6.5264,B 24.8565,C -2.7636,E1 25.1598,E2 89.9562} C_DIS
LIN {X 47.6722,Y 2.1268,Z 66,A -3.545,B 24.8558,C -2.7705,E1 25.1596,E2 86.9762} C_DIS
LIN {X 47.5777,Y 3.6788,Z 66,A -1.4061,B 24.8547,C -2.7816,E1 25.1591,E2 84.8236} C_DIS
LIN {X 47.3453,Y 5.9682,Z 66,A 1.2185,B 24.854,C -2.7875,E1 25.1583,E2 82.2007} C_DIS
LIN {X 47.0478,Y 7.9802,Z 66,A 3.7392,B 24.8531,C -2.7965,E1 25.1572,E2 79.6735} C_DIS
LIN {X 46.5458,Y 10.519,Z 66,A 6.7565,B 24.8523,C -2.8042,E1 25.1554,E2 76.6555} C_DIS
LIN {X 46.1485,Y 12.1447,Z 66,A 9.0246,B 24.8511,C -2.8152,E1 25.1538,E2 74.3743} C_DIS
LIN {X 44.9671,Y 15.973,Z 66,A 13.1757,B 24.851,C -2.8165,E1 25.1503,E2 70.2438} C_DIS
LIN {X 44.3358,Y 17.6495,Z 66,A 16.2274,B 24.8485,C -2.8401,E1 25.1472,E2 67.1533} C_DIS
LIN {X 43.2241,Y 20.2201,Z 66,A 18.762,B 24.8492,C -2.8334,E1 25.1443,E2 64.6482} C_DIS
LIN {X 41.8041,Y 23.014,Z 66,A 23.6652,B 24.8457,C -2.8655,E1 25.1378,E2 59.695} C_DIS
LIN {X 39.8954,Y 26.1827,Z 66,A 27.4468,B 24.8459,C -2.8641,E1 25.1322,E2 55.9357} C_DIS
LIN {X 37.8275,Y 29.0903,Z 66,A 31.5169,B 24.8452,C -2.8704,E1 25.1255,E2 51.8703} C_DIS
LIN {X 35.7261,Y 31.6362,Z 66,A 34.9914,B 24.8452,C -2.8702,E1 25.1192,E2 48.4121} C_DIS
LIN {X 33.8819,Y 33.6034,Z 66,A 38.6759,B 24.8436,C -2.8854,E1 25.1121,E2 44.7075} C_DIS
LIN {X 31.7487,Y 35.6258,Z 66,A 42.5338,B 24.8421,C -2.8984,E1 25.1041,E2 40.8343} C_DIS
LIN {X 28.7311,Y 38.1012,Z 66,A 47.2421,B 24.8412,C -2.9072,E1 25.0938,E2 36.1227} C_DIS
LIN {X 25.398,Y 40.3991,Z 66,A 51.7282,B 24.8411,C -2.9081,E1 25.0834,E2 31.6495} C_DIS
LIN {X 23.584,Y 41.485,Z 66,A 54.3991,B 24.8404,C -2.914,E1 25.0769,E2 28.9727} C_DIS
LIN {X 20.9639,Y 42.8682,Z 66,A 57.4336,B 24.841,C -2.9092,E1 25.0694,E2 25.9578} C_DIS
LIN {X 19.6941,Y 43.4663,Z 66,A 59.6815,B 24.8397,C -2.921,E1 25.0637,E2 23.6877} C_DIS
LIN {X 17.4219,Y 44.4257,Z 66,A 62.493,B 24.8397,C -2.9213,E1 25.0564,E2 20.8817} C_DIS
LIN {X 14.8834,Y 45.3394,Z 66,A 65.7137,B 24.8394,C -2.9237,E1 25.0479,E2 17.6617} C_DIS
LIN {X 11.4738,Y 46.3199,Z 66,A 70.2735,B 24.8385,C -2.9315,E1 25.0356,E2 13.0907} C_DIS
LIN {X 7.1616,Y 47.1791,Z 66,A 75.6422,B 24.8381,C -2.9348,E1 25.0208,E2 7.7197} C_DIS
LIN {X 4.2469,Y 47.5302,Z 66,A 78.5432,B 24.8392,C -2.925,E1 25.0128,E2 4.8442} C_DIS
LIN {X 1.653,Y 47.691,Z 66,A 81.8966,B 24.8388,C -2.9286,E1 25.0034,E2 1.4831} C_DIS
LIN {X -0.479,Y 47.7174,Z 66,A 84.051,B 24.8396,C -2.9216,E1 24.9975,E2 -0.6545} C_DIS
LIN {X -3.0304,Y 47.6235,Z 66,A 87.9499,B 24.8382,C -2.9339,E1 24.9865,E2 -4.5836} C_DIS
LIN {X -6.3848,Y 47.2904,Z 66,A 91.782,B 24.8389,C -2.9282,E1 24.9759,E2 -8.4047} C_DIS
LIN {X -9.6241,Y 46.7391,Z 66,A 95.3248,B 24.8399,C -2.9189,E1 24.9662,E2 -11.929} C_DIS
LIN {X -11.6684,Y 46.271,Z 66,A 98.4596,B 24.8391,C -2.926,E1 24.9577,E2 -15.0852} C_DIS
LIN {X -14.2262,Y 45.5499,Z 66,A 101.5697,B 24.8396,C -2.9213,E1 24.9494,E2 -18.1893} C_DIS
LIN {X -17.559,Y 44.3718,Z 66,A 104.9817,B 24.8416,C -2.9034,E1 24.9406,E2 -21.5657} C_DIS
LIN {X -19.1506,Y 43.7078,Z 66,A 107.443,B 24.8413,C -2.9063,E1 24.9342,E2 -24.0395} C_DIS
LIN {X -21.2757,Y 42.7143,Z 66,A 110.2791,B 24.8417,C -2.9022,E1 24.9271,E2 -26.8733} C_DIS
LIN {X -23.5146,Y 41.5242,Z 66,A 113.4097,B 24.8422,C -2.8983,E1 24.9194,E2 -30.0036} C_DIS
LIN {X -25.6412,Y 40.2456,Z 66,A 116.4376,B 24.8427,C -2.8936,E1 24.9122,E2 -33.0298} C_DIS
LIN {X -27.3372,Y 39.1134,Z 66,A 118.5371,B 24.8437,C -2.8839,E1 24.9074,E2 -35.113} C_DIS
LIN {X -29.4553,Y 37.5443,Z 66,A 122.286,B 24.8435,C -2.8857,E1 24.8991,E2 -38.8799} C_DIS
LIN {X -32.2842,Y 35.1409,Z 66,A 127.1678,B 24.844,C -2.8818,E1 24.8888,E2 -43.7717} C_DIS
LIN {X -34.8916,Y 32.5528,Z 66,A 131.6035,B 24.8451,C -2.8715,E1 24.8803,E2 -48.202} C_DIS
LIN {X -37.7586,Y 29.1798,Z 66,A 136.4243,B 24.8473,C -2.8511,E1 24.8718,E2 -52.9963} C_DIS
LIN {X -39.5788,Y 26.6584,Z 66,A 139.9018,B 24.8487,C -2.8376,E1 24.8663,E2 -56.4586} C_DIS
LIN {X -40.6456,Y 25.003,Z 66,A 142.9534,B 24.8484,C -2.8403,E1 24.8617,E2 -59.5324} C_DIS
LIN {X -42.7885,Y 21.1261,Z 66,A 147.5103,B 24.8512,C -2.8148,E1 24.8558,E2 -64.0525} C_DIS
LIN {X -43.4453,Y 19.7403,Z 66,A 150.0041,B 24.8508,C -2.8181,E1 24.8529,E2 -66.5678} C_DIS
LIN {X -44.8173,Y 16.3883,Z 66,A 153.9615,B 24.8527,C -2.7999,E1 24.8489,E2 -70.5037} C_DIS
LIN {X -45.6819,Y 13.7954,Z 66,A 157.4373,B 24.8535,C -2.7924,E1 24.846,E2 -73.9817} C_DIS
LIN {X -46.414,Y 11.086,Z 66,A 160.8815,B 24.8545,C -2.783,E1 24.8436,E2 -77.4235} C_DIS
LIN {X -46.9934,Y 8.2944,Z 66,A 164.149,B 24.8559,C -2.7703,E1 24.8419,E2 -80.6797} C_DIS
LIN {X -47.3702,Y 5.7648,Z 66,A 167.007,B 24.8571,C -2.7578,E1 24.8408,E2 -83.5251} C_DIS
LIN {X -47.5586,Y 3.9193,Z 66,A 169.9857,B 24.8568,C -2.7608,E1 24.8401,E2 -86.5287} C_DIS
LIN {X -47.7182,Y -0.1758,Z 66,A 174.9678,B 24.8584,C -2.7461,E1 24.8398,E2 -91.5057} C_DIS
LIN {X -47.5107,Y -4.4614,Z 66,A -179.6259,B 24.8597,C -2.7335,E1 24.8409,E2 -96.9143} C_DIS
LIN {X -46.8809,Y -8.9076,Z 66,A -174.9433,B 24.8623,C -2.7074,E1 24.843,E2 -101.5624} C_DIS
LIN {X -46.0868,Y -12.3763,Z 66,A -170.955,B 24.864,C -2.6908,E1 24.8456,E2 -105.5343} C_DIS
LIN {X -45.3752,Y -14.7724,Z 66,A -167.7339,B 24.8646,C -2.6849,E1 24.8482,E2 -108.7598} C_DIS
LIN {X -44.6579,Y -16.818,Z 66,A -165.3553,B 24.8657,C -2.6744,E1 24.8505,E2 -111.1267} C_DIS
LIN {X -43.7316,Y -19.0976,Z 66,A -162.3054,B 24.8664,C -2.6673,E1 24.8537,E2 -114.1767} C_DIS
LIN {X -43.1485,Y -20.3807,Z 66,A -160.0762,B 24.8661,C -2.67,E1 24.8564,E2 -116.4246} C_DIS
LIN {X -41.5813,Y -23.4132,Z 66,A -156.6833,B 24.8682,C -2.6494,E1 24.8608,E2 -119.7861} C_DIS
LIN {X -40.4321,Y -25.346,Z 66,A -153.138,B 24.8677,C -2.6542,E1 24.866,E2 -123.361} C_DIS
LIN {X -39.0719,Y -27.3968,Z 66,A -149.7405,B 24.8678,C -2.6532,E1 24.8715,E2 -126.7729} C_DIS
LIN {X -37.1492,Y -29.9519,Z 66,A -146.3897,B 24.8694,C -2.6372,E1 24.8772,E2 -130.1014} C_DIS
LIN {X -35.0777,Y -32.3534,Z 66,A -142.266,B 24.8698,C -2.6334,E1 24.8849,E2 -134.2344} C_DIS
LIN {X -32.4034,Y -35.0318,Z 66,A -138.5523,B 24.8719,C -2.6122,E1 24.8923,E2 -137.9128} C_DIS
LIN {X -30.8451,Y -36.4111,Z 66,A -135.5527,B 24.8716,C -2.6148,E1 24.8986,E2 -140.9303} C_DIS
LIN {X -29.3893,Y -37.5965,Z 66,A -132.5589,B 24.8709,C -2.6218,E1 24.9053,E2 -143.9519} C_DIS
LIN {X -26.4257,Y -39.7352,Z 66,A -128.7585,B 24.8725,C -2.606,E1 24.914,E2 -147.7273} C_DIS
LIN {X -23.5783,Y -41.4879,Z 66,A -125.0325,B 24.8735,C -2.5959,E1 24.9229,E2 -151.4407} C_DIS
LIN {X -20.7819,Y -42.9566,Z 66,A -121.5922,B 24.8745,C -2.5859,E1 24.9314,E2 -154.8664} C_DIS
LIN {X -19.1686,Y -43.7006,Z 66,A -118.5318,B 24.8733,C -2.598,E1 24.9393,E2 -157.9629} C_DIS
LIN {X -16.5148,Y -44.7708,Z 66,A -115.2415,B 24.8738,C -2.5926,E1 24.9479,E2 -161.2473} C_DIS
LIN {X -13.1683,Y -45.8668,Z 66,A -111.5996,B 24.875,C -2.5802,E1 24.9576,E2 -164.8661} C_DIS
LIN {X -10.3704,Y -46.579,Z 66,A -107.6095,B 24.8744,C -2.5869,E1 24.9685,E2 -168.8774} C_DIS
LIN {X -7.8593,Y -47.068,Z 66,A -105.0775,B 24.8753,C -2.5771,E1 24.9754,E2 -171.3886} C_DIS
LIN {X -6.1077,Y -47.3271,Z 66,A -102.189,B 24.8741,C -2.5892,E1 24.9834,E2 -174.3082} C_DIS
LIN {X -2.5377,Y -47.652,Z 66,A -98.6352,B 24.8754,C -2.5767,E1 24.9933,E2 -177.8337} C_DIS
LIN {X -0.4066,Y -47.7181,Z 66,A -95.8452,B 24.8749,C -2.581,E1 25.0011,E2 -180.6341} C_DIS
LIN {X -0.4066,Y -47.7181,Z 66,A -95.8452,B 24.8749,C -2.581,E1 25.0011,E2 -180.6341} C_DIS
Enddeposition()
LIN {X 0.2144,Y -46.7557,Z 66,A -95.048,B 24.8732,C -2.5985,E1 25.0034,E2 -181.4728} C_DIS
Startdeposition()
$VEL.CP = VEL_PRINT
LIN {X -1.8495,Y -46.7243,Z 66,A -99.207,B 24.8759,C -2.5715,E1 24.9916,E2 -177.2494} C_DIS
LIN {X -4.8629,Y -46.507,Z 66,A -102.9461,B 24.8759,C -2.5711,E1 24.9812,E2 -173.5075} C_DIS
LIN {X -6.8216,Y -46.2608,Z 66,A -105.1167,B 24.8755,C -2.5754,E1 24.9752,E2 -171.3456} C_DIS
LIN {X -9.263,Y -45.834,Z 66,A -108.4283,B 24.8758,C -2.5723,E1 24.9661,E2 -168.0229} C_DIS
LIN {X -12.3329,Y -45.1051,Z 66,A -112.6962,B 24.8762,C -2.5684,E1 24.9545,E2 -163.7395} C_DIS
LIN {X -15.7151,Y -44.0409,Z 66,A -116.3528,B 24.8748,C -2.5821,E1 24.9449,E2 -160.1087} C_DIS
LIN {X -19.5225,Y -42.4902,Z 66,A -121.706,B 24.8748,C -2.5825,E1 24.9311,E2 -154.7443} C_DIS
LIN {X -22.0142,Y -41.2552,Z 66,A -124.8549,B 24.874,C -2.5905,E1 24.9233,E2 -151.6058} C_DIS
LIN {X -24.2417,Y -39.9862,Z 66,A -128.5885,B 24.8744,C -2.5864,E1 24.9143,E2 -147.8513} C_DIS
LIN {X -26.2225,Y -38.7161,Z 66,A -132.0485,B 24.8748,C -2.5829,E1 24.9063,E2 -144.3713} C_DIS
LIN {X -28.9883,Y -36.6911,Z 66,A -135.9181,B 24.8736,C -2.5948,E1 24.8978,E2 -140.5158} C_DIS
LIN {X -31.7232,Y -34.3543,Z 66,A -139.8425,B 24.8721,C -2.6099,E1 24.8896,E2 -136.6118} C_DIS
LIN {X -33.9958,Y -32.1068,Z 66,A -143.3079,B 24.8707,C -2.6242,E1 24.8829,E2 -133.1659} C_DIS
LIN {X -35.4993,Y -30.4365,Z 66,A -146.4433,B 24.8707,C -2.6251,E1 24.877,E2 -130.0186} C_DIS
LIN {X -37.0863,Y -28.4809,Z 66,A -149.9418,B 24.8704,C -2.6268,E1 24.871,E2 -126.5076} C_DIS
LIN {X -38.7617,Y -26.1552,Z 66,A -154.0065,B 24.8703,C -2.6283,E1 24.8646,E2 -122.4263} C_DIS
LIN {X -40.7502,Y -22.9348,Z 66,A -157.7268,B 24.8679,C -2.6522,E1 24.8594,E2 -118.7439} C_DIS
LIN {X -41.8993,Y -20.7605,Z 66,A -160.6961,B 24.867,C -2.6609,E1 24.8556,E2 -115.7795} C_DIS
LIN {X -42.8211,Y -18.7862,Z 66,A -163.445,B 24.8664,C -2.6673,E1 24.8525,E2 -113.0308} C_DIS
LIN {X -43.643,Y -16.7877,Z 66,A -165.7598,B 24.8652,C -2.6791,E1 24.8501,E2 -110.7313} C_DIS
LIN {X -44.4362,Y -14.5596,Z 66,A -169.2824,B 24.8652,C -2.6795,E1 24.8469,E2 -107.1897} C_DIS
LIN {X -45.1318,Y -12.2339,Z 66,A -171.9872,B 24.8639,C -2.6918,E1 24.8448,E2 -104.4984} C_DIS
LIN {X -45.701,Y -9.8985,Z 66,A -174.7398,B 24.8628,C -2.7031,E1 24.8431,E2 -101.7567} C_DIS
LIN {X -46.0551,Y -8.093,Z 66,A -177.1856,B 24.8623,C -2.7075,E1 24.8419,E2 -99.307} C_DIS
LIN {X -46.4692,Y -5.2136,Z 66,A 179.1762,B 24.8613,C -2.7176,E1 24.8406,E2 -95.6712} C_DIS
LIN {X -46.6364,Y -3.4152,Z 66,A 176.8948,B 24.8607,C -2.7236,E1 24.8401,E2 -93.3905} C_DIS
LIN {X -46.7519,Y -0.9018,Z 66,A 173.8821,B 24.8596,C -2.7341,E1 24.8398,E2 -90.3848} C_DIS
LIN {X -46.7335,Y 1.5934,Z 66,A 170.4889,B 24.859,C -2.7396,E1 24.84,E2 -86.9842} C_DIS
LIN {X -46.5251,Y 4.6885,Z 66,A 167.2348,B 24.8571,C -2.7583,E1 24.8407,E2 -83.7554} C_DIS
LIN {X -46.2544,Y 6.8656,Z 66,A 164.2192,B 24.8566,C -2.7627,E1 24.8419,E2 -80.7322} C_DIS
LIN {X -45.9351,Y 8.7473,Z 66,A 161.4997,B 24.8564,C -2.7653,E1 24.8433,E2 -78.0028} C_DIS
LIN {X -45.1373,Y 12.214,Z 66,A 157.5475,B 24.8544,C -2.7838,E1 24.8459,E2 -74.0719} C_DIS
LIN {X -44.4408,Y 14.5451,Z 66,A 154.7217,B 24.8533,C -2.7949,E1 24.8482,E2 -71.2562} C_DIS
LIN {X -43.8658,Y 16.197,Z 66,A 152.2552,B 24.853,C -2.7973,E1 24.8506,E2 -68.7816} C_DIS
LIN {X -42.6183,Y 19.2415,Z 66,A 148.4241,B 24.8515,C -2.8118,E1 24.8547,E2 -64.9639} C_DIS
LIN {X -41.7347,Y 21.0893,Z 66,A 146.0104,B 24.8506,C -2.8203,E1 24.8577,E2 -62.5575} C_DIS
LIN {X -40.6538,Y 23.1056,Z 66,A 142.8125,B 24.8503,C -2.8232,E1 24.862,E2 -59.3498} C_DIS
LIN {X -39.14,Y 25.586,Z 66,A 139.1655,B 24.8493,C -2.8319,E1 24.8674,E2 -55.7052} C_DIS
LIN {X -37.6748,Y 27.6979,Z 66,A 136.3042,B 24.848,C -2.8441,E1 24.8721,E2 -52.8588} C_DIS
LIN {X -36.1441,Y 29.6683,Z 66,A 132.9383,B 24.8476,C -2.8479,E1 24.8779,E2 -49.4864} C_DIS
LIN {X -34.5011,Y 31.5632,Z 66,A 130.1066,B 24.8465,C -2.8587,E1 24.8832,E2 -46.6678} C_DIS
LIN {X -33.0553,Y 33.0752,Z 66,A 127.5637,B 24.8458,C -2.865,E1 24.8881,E2 -44.1292} C_DIS
LIN {X -31.2313,Y 34.8018,Z 66,A 124.2038,B 24.8454,C -2.8683,E1 24.895,E2 -40.7634} C_DIS
LIN {X -29.1404,Y 36.5708,Z 66,A 120.9342,B 24.8445,C -2.8766,E1 24.9021,E2 -37.5013} C_DIS
LIN {X -27.0635,Y 38.133,Z 66,A 117.7896,B 24.8438,C -2.8836,E1 24.9091,E2 -34.3622} C_DIS
LIN {X -24.1527,Y 40.0399,Z 66,A 112.6959,B 24.8441,C -2.8801,E1 24.9212,E2 -29.2442} C_DIS
LIN {X -21.2154,Y 41.6708,Z 66,A 108.9816,B 24.8428,C -2.8923,E1 24.9304,E2 -25.5488} C_DIS
LIN {X -17.9896,Y 43.1616,Z 66,A 105.0734,B 24.8414,C -2.9049,E1 24.9403,E2 -21.6612} C_DIS
LIN {X -15.7998,Y 44.0105,Z 66,A 101.8121,B 24.8416,C -2.9031,E1 24.9489,E2 -18.389} C_DIS
LIN {X -13.4313,Y 44.7902,Z 66,A 98.8817,B 24.8411,C -2.9083,E1 24.9567,E2 -15.4659} C_DIS
LIN {X -10.7141,Y 45.5163,Z 66,A 95.9375,B 24.8399,C -2.919,E1 24.9646,E2 -12.5429} C_DIS
LIN {X -9.3811,Y 45.8099,Z 66,A 93.8126,B 24.8405,C -2.9137,E1 24.9704,E2 -10.4028} C_DIS
LIN {X -6.1249,Y 46.3578,Z 66,A 90.0536,B 24.8397,C -2.9207,E1 24.9808,E2 -6.6572} C_DIS
LIN {X -3.5253,Y 46.6276,Z 66,A 86.5032,B 24.8401,C -2.917,E1 24.9907,E2 -3.0961} C_DIS
LIN {X -0.6992,Y 46.7555,Z 66,A 82.8456,B 24.8403,C -2.915,E1 25.0009,E2 0.5666} C_DIS
LIN {X 2.8097,Y 46.6767,Z 66,A 79.2101,B 24.8392,C -2.9257,E1 25.011,E2 4.1758} C_DIS
LIN {X 4.2319,Y 46.5685,Z 66,A 77.2059,B 24.8396,C -2.9216,E1 25.0166,E2 6.1888} C_DIS
LIN {X 6.2965,Y 46.3339,Z 66,A 74.6104,B 24.8397,C -2.9203,E1 25.0237,E2 8.7853} C_DIS
LIN {X 9.2441,Y 45.8379,Z 66,A 70.3018,B 24.841,C -2.9086,E1 25.0356,E2 13.1167} C_DIS
LIN {X 12.8448,Y 44.9619,Z 66,A 66.3302,B 24.8403,C -2.915,E1 25.0463,E2 17.0669} C_DIS
LIN {X 15.2597,Y 44.2006,Z 66,A 63.1353,B 24.8408,C -2.911,E1 25.0548,E2 20.2653} C_DIS
LIN {X 19.2228,Y 42.6268,Z 66,A 58.1388,B 24.8409,C -2.9095,E1 25.0676,E2 25.2538} C_DIS
LIN {X 21.7228,Y 41.4085,Z 66,A 54.1832,B 24.8424,C -2.896,E1 25.0775,E2 29.2305} C_DIS
LIN {X 23.8917,Y 40.1964,Z 66,A 50.7232,B 24.8437,C -2.8846,E1 25.0859,E2 32.7069} C_DIS
LIN {X 26.7041,Y 38.3855,Z 66,A 47.3714,B 24.843,C -2.8909,E1 25.0936,E2 36.0326} C_DIS
LIN {X 29.1167,Y 36.5895,Z 66,A 44.2714,B 24.8426,C -2.8946,E1 25.1004,E2 39.1124} C_DIS
LIN {X 30.457,Y 35.4814,Z 66,A 41.7941,B 24.8437,C -2.8846,E1 25.1057,E2 41.6041} C_DIS
LIN {X 32.2835,Y 33.8285,Z 66,A 38.9759,B 24.8439,C -2.8821,E1 25.1115,E2 44.4166} C_DIS
LIN {X 34.1005,Y 31.9953,Z 66,A 35.8209,B 24.8446,C -2.8756,E1 25.1177,E2 47.5735} C_DIS
LIN {X 36.0463,Y 29.7865,Z 66,A 32.0096,B 24.8459,C -2.8638,E1 25.1246,E2 51.3955} C_DIS
LIN {X 37.1583,Y 28.3876,Z 66,A 29.712,B 24.8467,C -2.8567,E1 25.1286,E2 53.6991} C_DIS
LIN {X 38.8118,Y 26.0807,Z 66,A 26.4511,B 24.8472,C -2.852,E1 25.1338,E2 56.9549} C_DIS
LIN {X 40.2313,Y 23.8327,Z 66,A 22.8448,B 24.8488,C -2.8373,E1 25.139,E2 60.5779} C_DIS
LIN {X 42.0067,Y 20.5426,Z 66,A 18.2095,B 24.8502,C -2.8239,E1 25.145,E2 65.2202} C_DIS
Enddeposition()
END
